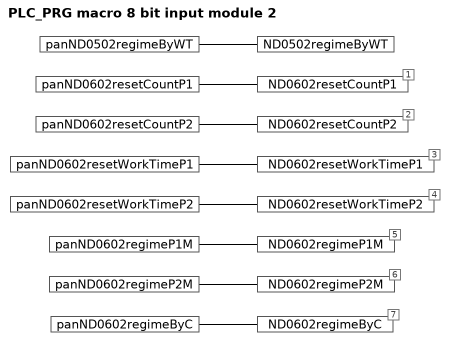
[picture p72: PLC_PRG macro 8 bit input module 2 (CFC)]
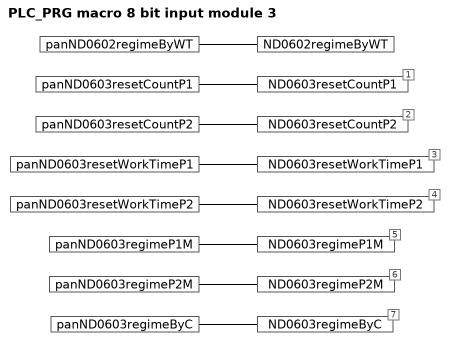
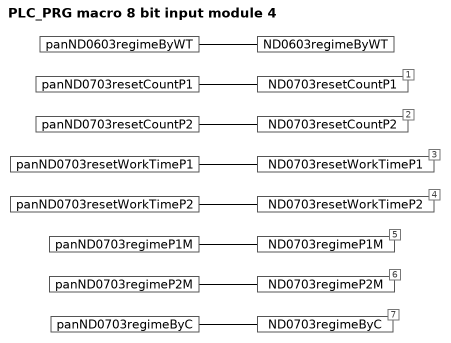
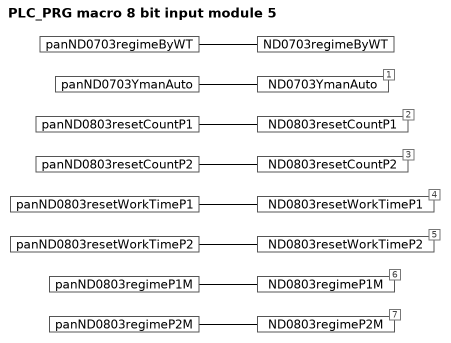
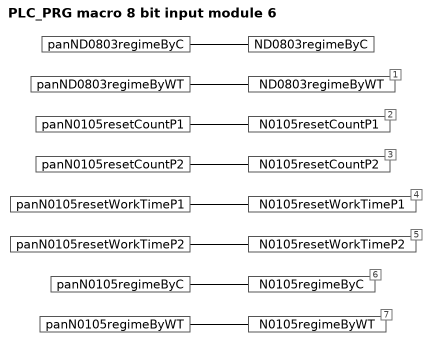
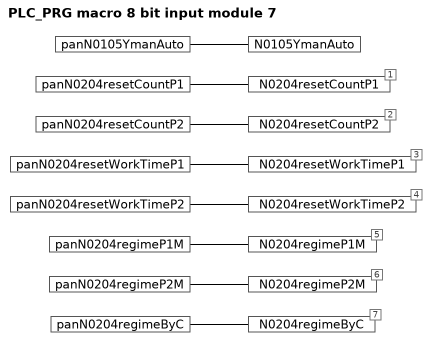
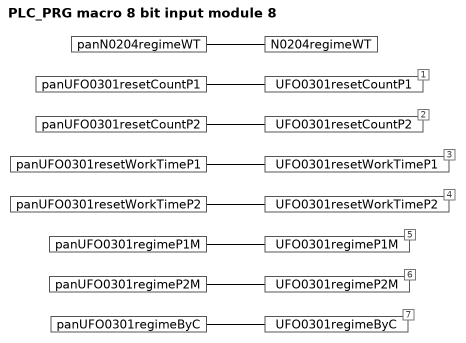
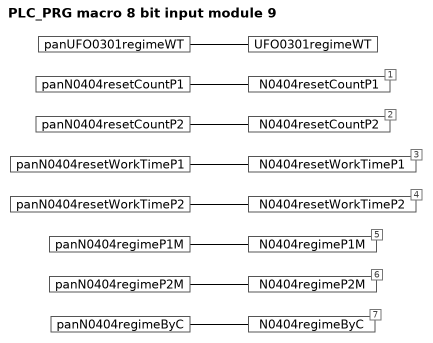
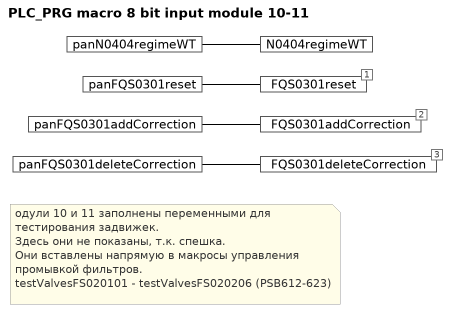
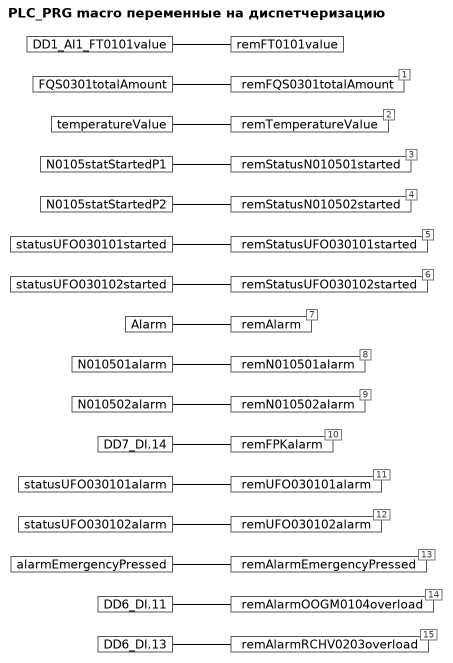
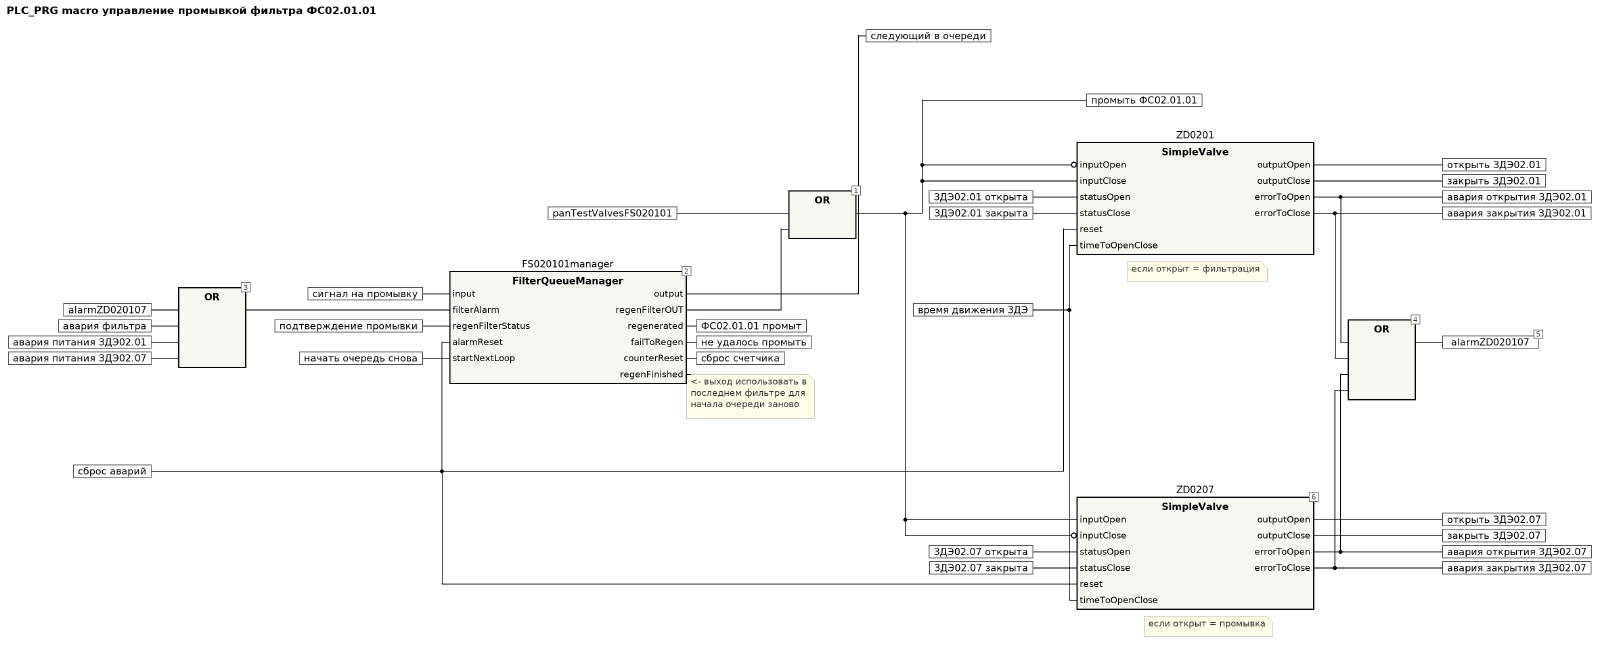
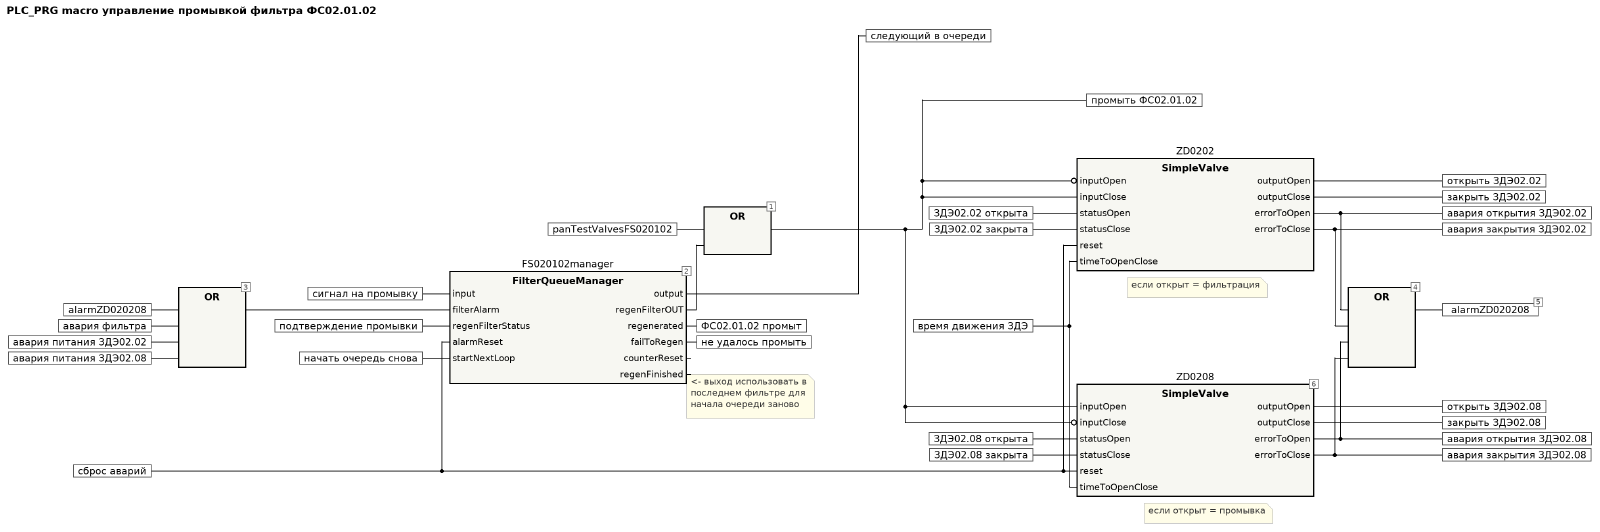
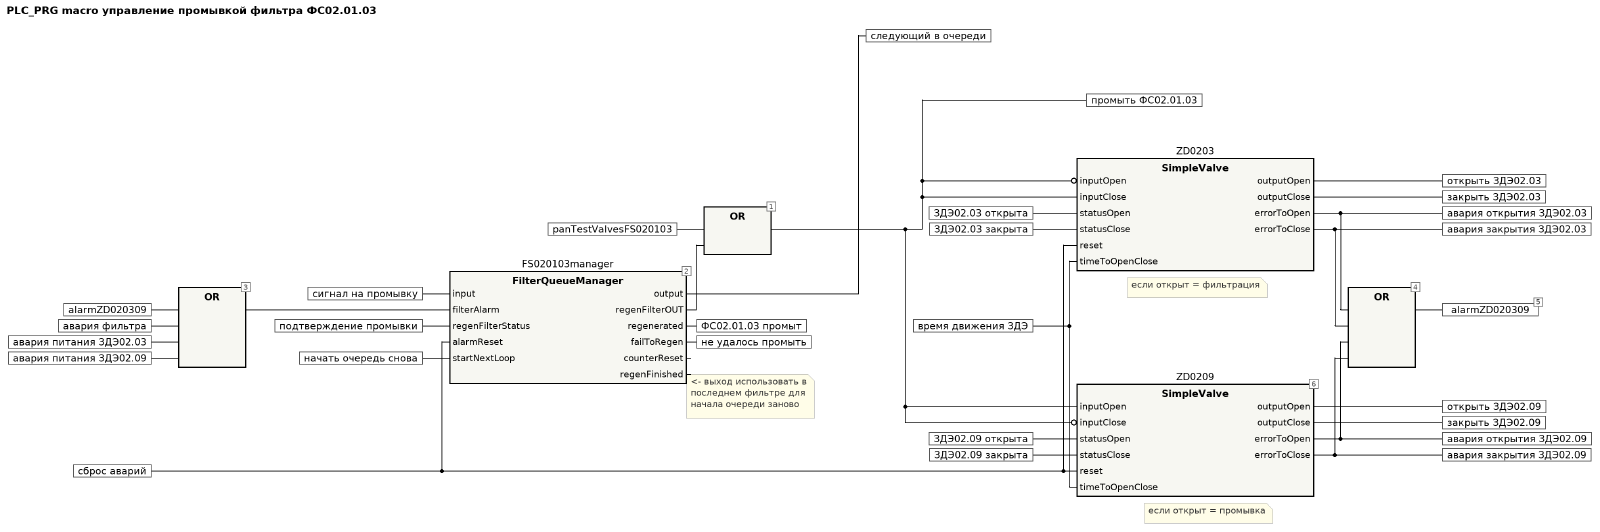
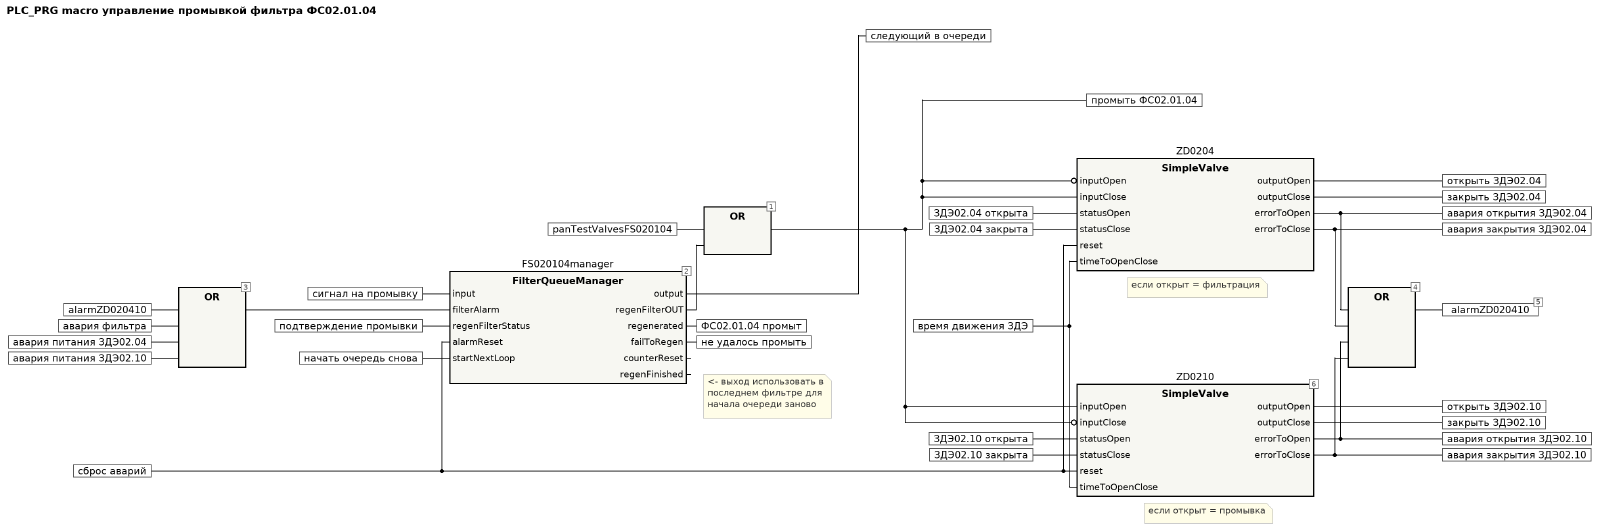
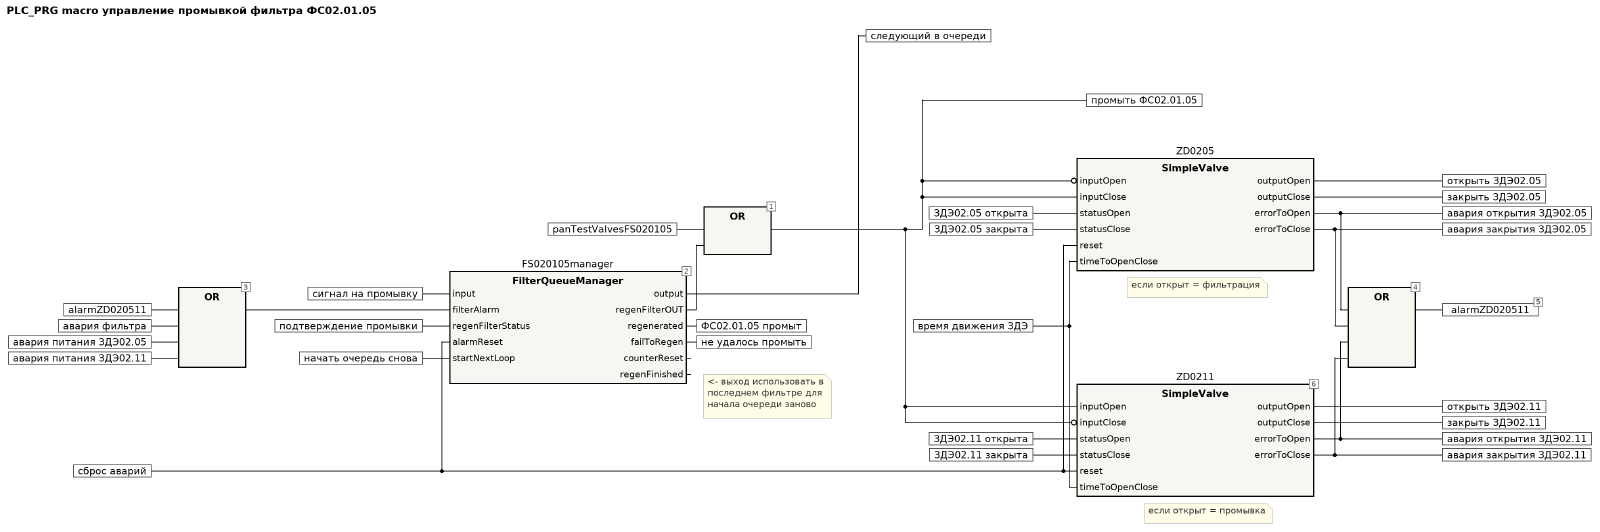
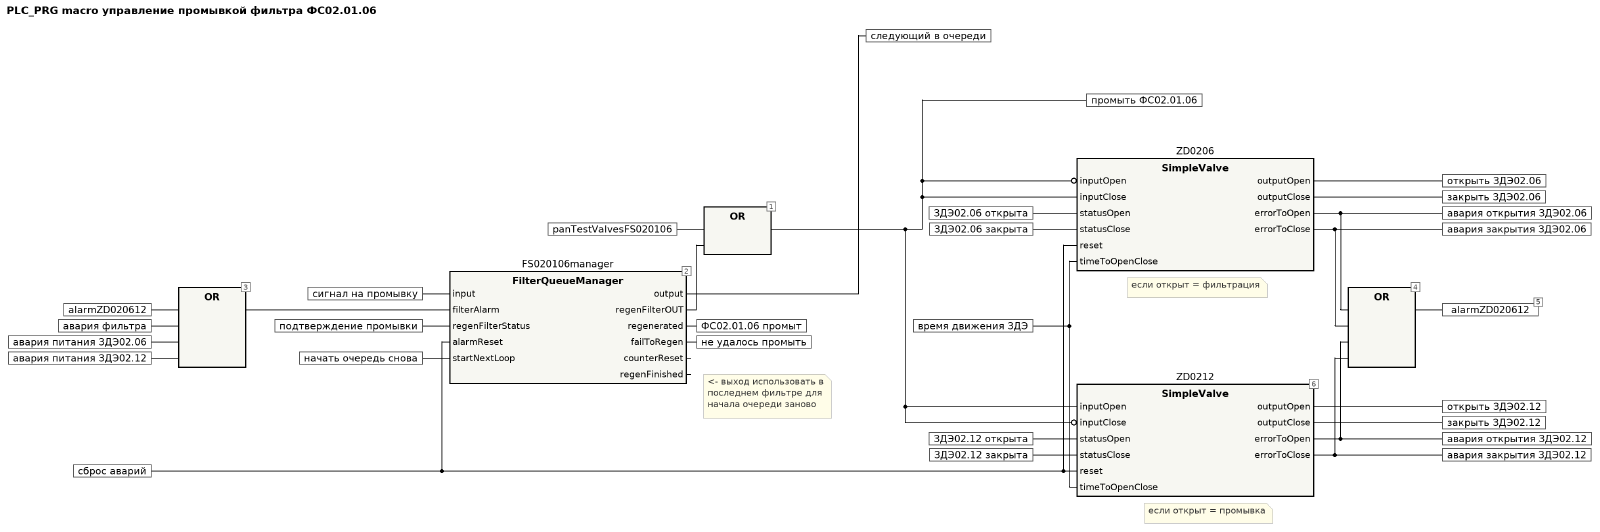
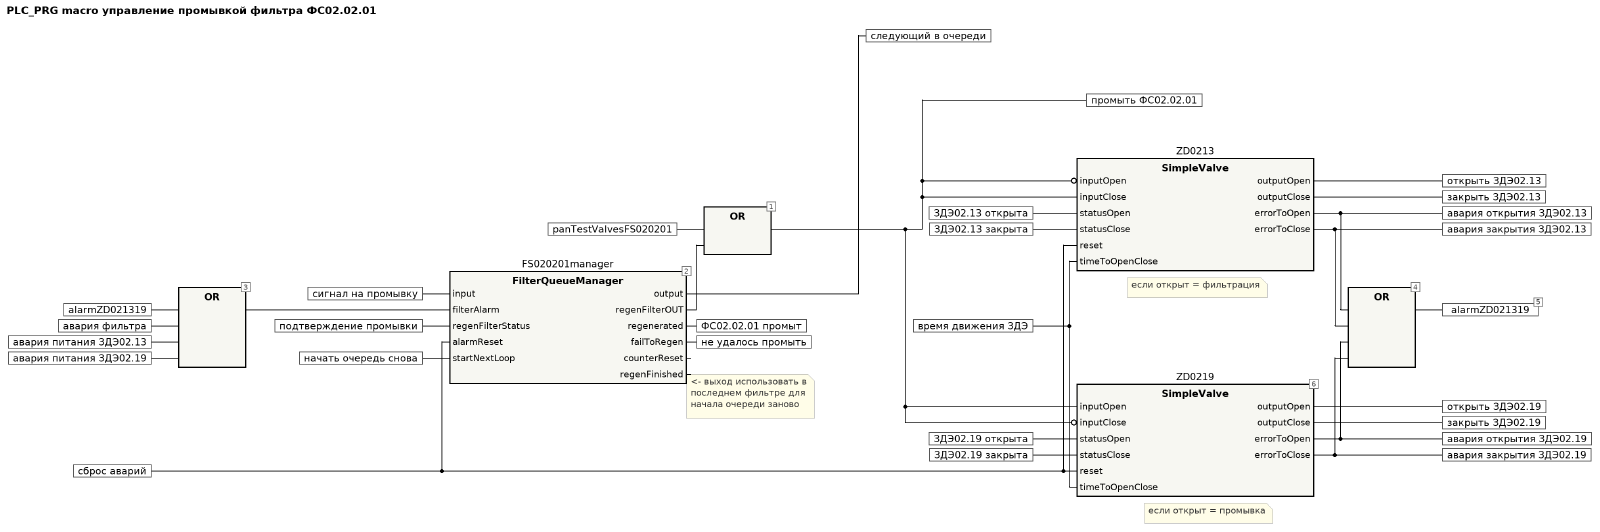
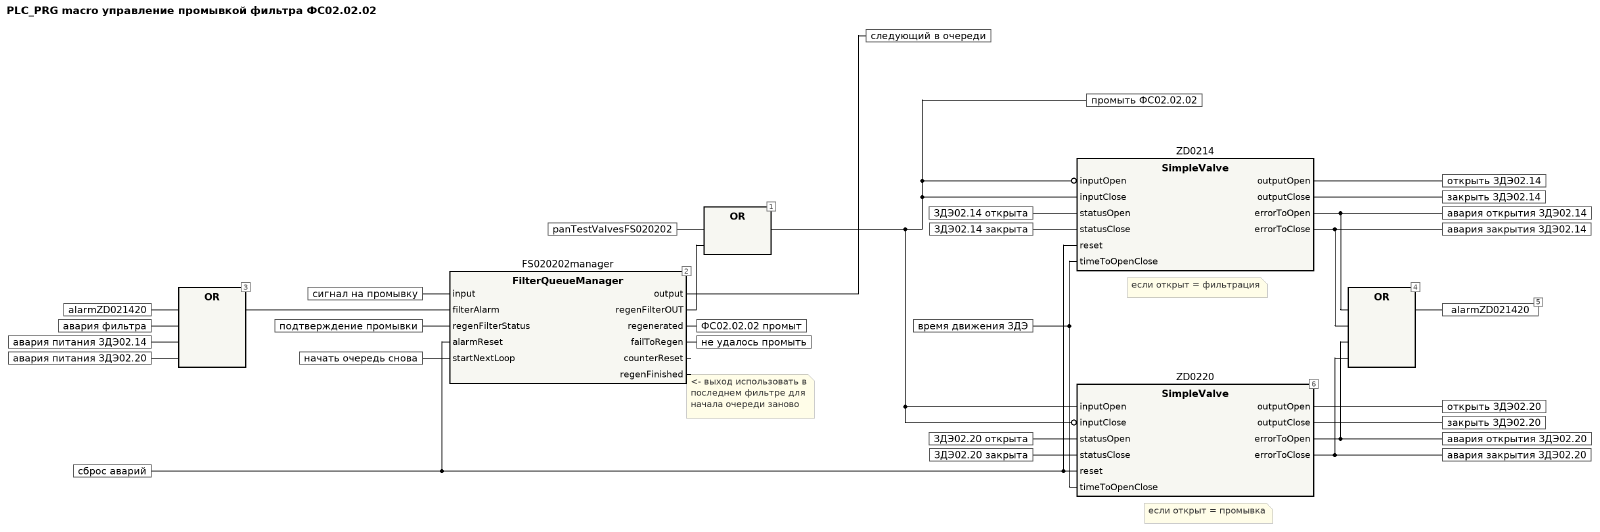
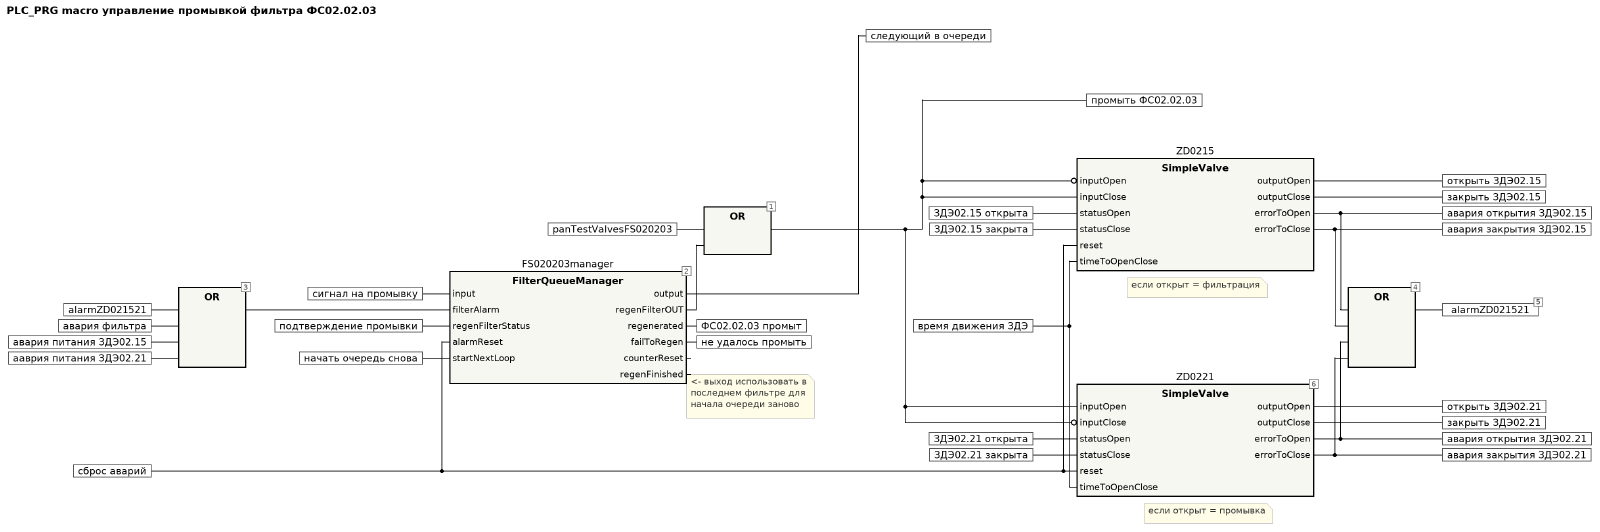
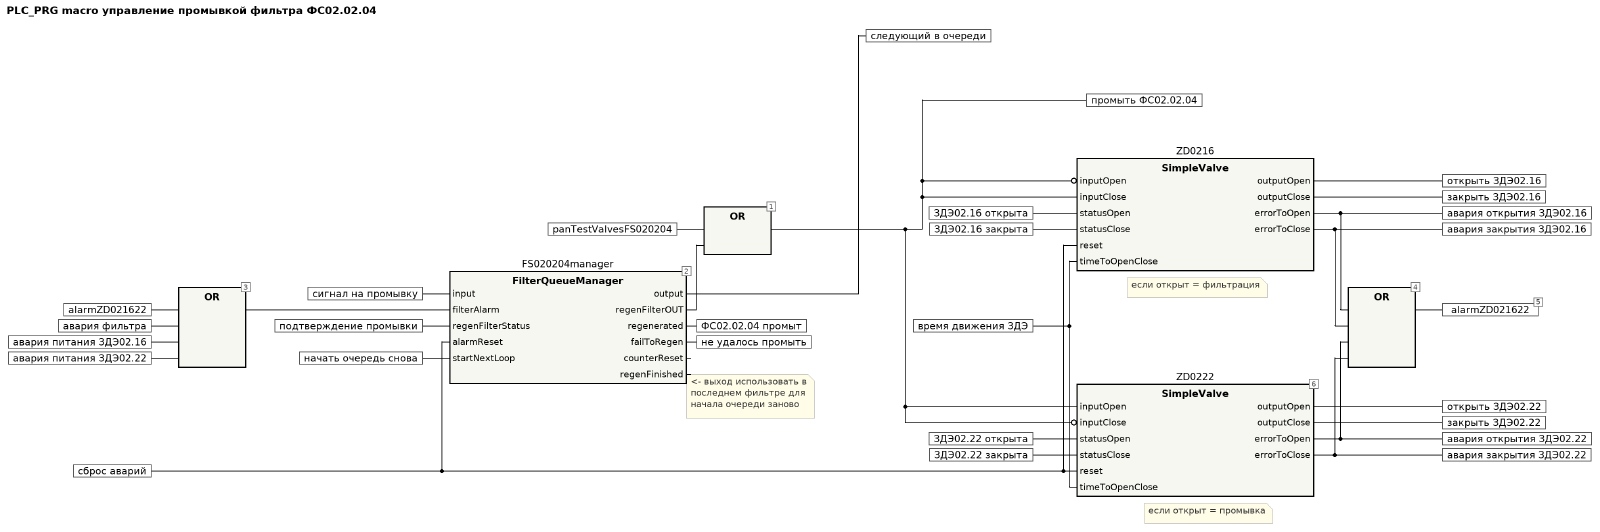
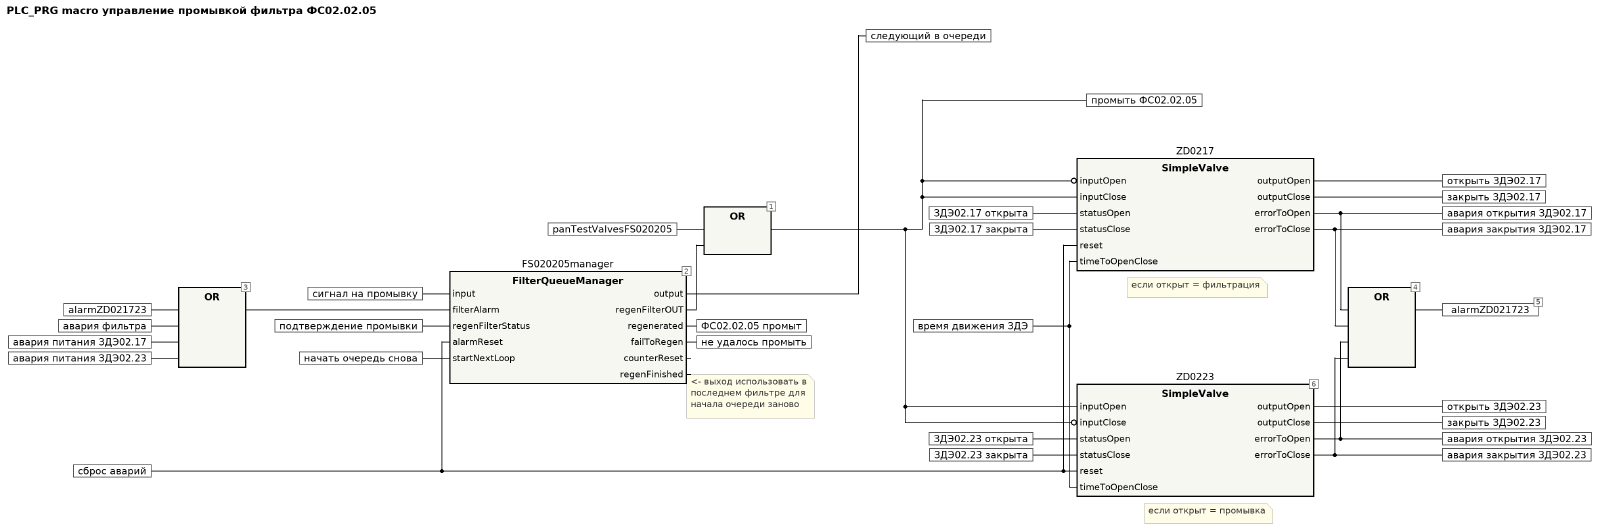
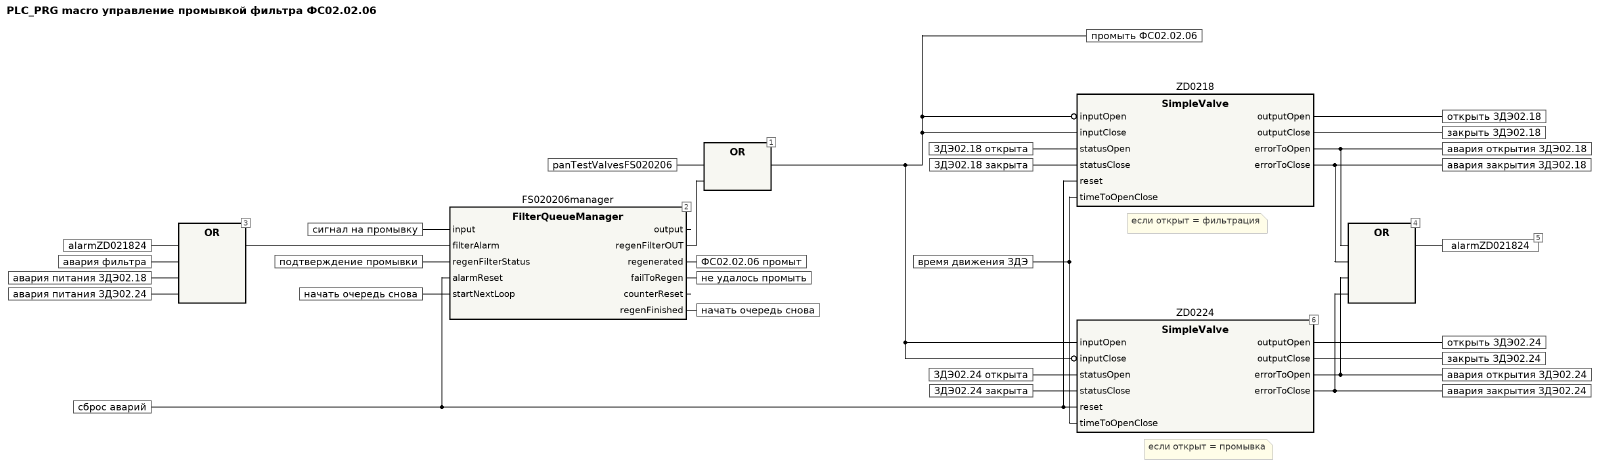
_CFC_ (* Continuous Function Chart, elements in execution order *)
(* в этом макросе лежит управление режимом тестирования задвижек ЗДЭ03 / Тестирование запрещает автоматический запуск УФО от ПЛК *)
(* 1=открыть; 0 = закрыть *)
(* авария питания КШЭ04.01 *)
(* авария НД05.02/02 *)
(* авария НД05.02/01 *)
(* инвертирование сигнала, чтобы все аварии / обозначались как 1 (TRUE) *)
(* авария питания ЗДЭ02.24 *)
(* авария питания ЗДЭ02.23 *)
(* авария питания ЗДЭ02.22 *)
(* авария питания ЗДЭ02.21 *)
(* авария питания ЗДЭ02.20 *)
(* авария питания ЗДЭ02.19 *)
(* авария питания ЗДЭ02.18 *)
(* авария питания ЗДЭ02.17 *)
(* авария питания ЗДЭ02.16 *)
(* авария питания ЗДЭ02.15 *)
(* авария питания ЗДЭ02.14 *)
(* авария питания ЗДЭ02.13 *)
(* авария питания ЗДЭ02.12 *)
(* авария питания ЗДЭ02.11 *)
(* авария питания ЗДЭ02.10 *)
(* авария питания ЗДЭ02.09 *)
(* авария питания ЗДЭ02.08 *)
(* авария питания ЗДЭ02.07 *)
(* авария питания ЗДЭ02.06 *)
(* авария питания ЗДЭ02.05 *)
(* авария питания ЗДЭ02.04 *)
(* авария питания ЗДЭ02.03 *)
(* авария питания ЗДЭ02.02 *)
(* авария питания ЗДЭ02.01 *)
(* очередь передается на 2 ступень *)
(* подсчет общего объема стоков, прошедшего через расходомер FT01.02 *)
(* сброс счетчика стоков до следующей промывки *)
(* авария (при 0) ФС02.02/01 *)
(* авария (при 0) ФС02.02/02 *)
(* авария (при 0) ФС02.02/03 *)
(* авария (при 0) ФС02.02/04 *)
(* авария (при 0) ФС02.02/05 *)
(* авария (при 0) ФС02.02/06 *)
(* авария (при 0) ФС02.01/01 *)
(* авария (при 0) ФС02.01/02 *)
(* авария (при 0) ФС02.01/03 *)
(* авария (при 0) ФС02.01/04 *)
(* авария (при 0) ФС02.01/05 *)
(* авария (при 0) ФС02.01/06 *)
(* 0=авария *)
(* заданный до промывки объем *)
(* текущий объем *)
(* Пуск Н02.04/02 *)
(* Пуск Н02.04/01 *)
(* Стоп Н02.04 *)
(* Сухой ход Н02.04 (LS02.03) 0=сух.ход *)
(* Клапан КЭМ08.01 открыт. *)
(* Клапан КЭМ07.01 открыт. *)
(* Клапан КЭМ06.01 открыт. *)
(* Клапан КЭМ05.01 открыт. *)
(* промывка ФС02.02/01 *)
(* промывка ФС02.02/02 *)
(* промывка ФС02.02/03 *)
(* промывка ФС02.02/04 *)
(* промывка ФС02.02/05 *)
(* промывка ФС02.02/06 *)
(* Авария Н02.04/02 (0=авария) *)
(* Авария Н02.04/01 (0=авария) *)
(* импульсный расходомер *)
(* авария Н04.04/02, 0=авария *)
(* авария Н04.04/01, 0=авария *)
(* сухой ход Н04.04, 0=защита *)
(* авт.пуск Н04.04 *)
(* пуск Н04.04/01 *)
(* пуск Н04.04/02 *)
(* стоп Н04.04 *)
(* подающий насос ФПК работает *)
(* статус КШЭ04.01 закрыт *)
(* Закрыть КШЭ04.01 *)
(* статус КШЭ04.01 открыт *)
(* Открыть КШЭ04.01 *)
(* авария ФПК *)
(* Авария входа AI6 ПЛК, давл.ФПК *)
(* Давление на входе ФПК / 0...16 бар (мах допуст.10) *)
(* LSА02.01 Перелив РЧВ02.03 *)
(* авария питания ЗДЭ02.25 *)
(* термоконтакт Н01.05/02 *)
(* термоконтакт Н01.05/01 *)
(* Авария ЧРП Н01.05 *)
(* КМ3 питание насоса 2 *)
(* КМ2 питание насоса 1 *)
(* КМ1 питание ЧРП *)
(* Пуск  Н01.05 *)
(* время на создание потока *)
(* Стоп  Н01.05 (сброс самоподхвата реле) *)
(* SA1 Ручной выбор Н01.05/02 = главный *)
(* SA1 Ручной выбор Н01.05/01 = главный *)
(* LS01.04 - нижний уровень ОГМ01.04, сухой ход Н01.05 *)
(* LS01.03 - рабочий верхний уровень ОГМ01.04 автоматический пуск 01.05 *)
(* Статус ПУСК ЧРП Н01.05 *)
(* Инициализирует требуемые булевые переменные / в момент старта выполнения программы. *)
(* LSA01.02 перелив ОГМ01.04 *)
(* сухой ход НД08.03/02 *)
(* сухой ход НД08.03/01 *)
(* сухой ход НД08.03/02 *)
(* сухой ход НД08.03/01 *)
(* авария входа рН-метра QE01.02 *)
(* рН-метр QE01.01 на входе, / диапазон 0...14 *)
(* расходомер FT01.02 на входе, / диапазон 0...600куб/час *)
(* авария входа расходомера FT01.01 *)
(* управление 4...20мА НД08.04 *)
(* пуск/стоп НД08.04 *)
(* насос Н04.01 работает *)
(* авария НД08.04 *)
(* авария привода НД08.03/02 *)
(* авария привода НД08.03/01 *)
(* АВАРИИ *)
(* управление 4...20мА НД05.02/02 *)
(* пуск/стоп НД05.02/02 *)
(* авария НД05.02/02 *)
(* авария НД05.02/01 *)
(* пуск/стоп НД05.02/01 *)
(* управление 4...20мА НД05.02/01 *)
(* датчик температуры в помещении / (метран) диапазон: 0...+100С *)
(* лампа АВАРИЯ *)
(* авария входа датчика температуры *)
(* ошибка блока дозирования НД05.02 *)
(* авария НД06.02/02 *)
(* авария НД06.02/01 *)
(* управление 4...20мА НД06.02/02 *)
(* пуск/стоп НД06.02/02 *)
(* пуск/стоп НД06.02/01 *)
(* управление 4...20мА НД06.02/01 *)
(* авария НД06.03/02 *)
(* авария НД06.03/01 *)
(* управление 4...20мА НД06.03/02 *)
(* пуск/стоп НД06.03/02 *)
(* пуск/стоп НД06.03/01 *)
(* управление 4...20мА НД06.03/01 *)
(* авария НД06.02/02 *)
(* авария НД06.02/01 *)
(* авария НД06.03/02 *)
(* авария НД06.03/01 *)
(* авария НД07.03/02 *)
(* авария НД07.03/01 *)
(* пуск/стоп НД07.03/02 *)
(* пуск/стоп НД07.03/01 *)
(* управление 4...20мА НД07.03/02 *)
(* управление 4...20мА НД07.03/01 *)
(* авария НД07.03/02 *)
(* авария НД07.03/01 *)
(* авария привода НД08.03/02 *)
(* авария привода НД08.03/01 *)
(* управление 4...20мА НД08.03/02 *)
(* пуск/стоп НД08.03/02 *)
(* пуск/стоп НД08.03/01 *)
(* управление 4...20мА НД08.03/01 *)
(* авария НД08.04 *)
(* расходомер FT01.01 на входе, / диапазон 0...600куб/час *)
(* авария входа расходомера FT01.02 *)
(* авария входа рН-метра QE01.01 *)
(* рН-метр QE01.02 на входе, / диапазон 0...14 *)
(* ФПК не запустился *)
(* ФПК готов к приему *)
(* подающий насос ФПК работает *)
(* авария ФПК *)
(* Давление на входе ФПК (0...16 бар) *)
(* датчик уровня осадка *)
(* Защита от сухого хода насоса ФПК *)
(* запуск фильтрации *)
(* время работы ФПК после спада сигнала датч.осадка *)
(* время контроля старта ФПК (по умолч.=3мин) *)
(* авария Н04.04/02 *)
(* авария Н04.04/01 *)
(* авария УФО03.01/01 *)
(* авария УФО03.01/02 *)
(* работа УФО03.01/01 *)
(* Для подачи предостережения на пульте / оператора (при необходимости), а также / сигнализации лампой АВАРИЯ. *)
(* авария УФО03.01/01 *)
(* работа УФО03.01/02 *)
(* авария УФО03.01/02 *)
(* Контроль, если УФО включили вручную, / а потока при этом нет. *)
(* работа М06.04 (УПК) *)
(* работа М07.02 (УПЩ) *)
(* работа М08.02 (УПФ) *)
(* авария М06.04 (УПК) *)
(* авария М07.02 (УПЩ) *)
(* авария М08.02 (УПФ) *)
(* пуск/стоп НД07.03/02 *)
(* пуск/стоп НД07.03/01 *)
(* пуск/стоп НД08.04 *)
(* пуск/стоп НД06.02/02 *)
(* пуск/стоп НД06.02/01 *)
(* пуск/стоп НД06.03/02 *)
(* пуск/стоп НД06.03/01 *)
(* пуск/стоп НД08.03/02 *)
(* пуск/стоп НД08.03/01 *)
(* промывка ФС02.01/01 *)
(* промывка ФС02.01/02 *)
(* промывка ФС02.01/03 *)
(* промывка ФС02.01/04 *)
(* промывка ФС02.01/05 *)
(* промывка ФС02.01/06 *)
(* Авария Н02.04/02 (0=авария) *)
(* Авария Н02.04/01 (0=авария) *)
(* здесь мгновенный расход / в кубометрах в час (FT01.02) *)
(* выдает импульс / каждую секунду *)
(* если есть расход / (больше нуля) *)
(* преобразуем расход из / кубометров в час в / кубометры в секунду *)
(* суммируем каждую секунду значение / мгновенного расхода в кубометрах в секунду *)
(* блок подачи сигнала на промывку *)
(* авария КНС *)
(* Авария питания розеток / управл.клапанов фильтров. *)
(* Авария питания клапанов КЭМ. *)
(* авария сети (РКФ) *)
(* Блок управления разрешением работы КНС *)
(* Нажат аварийный стоп. *)
(* разрешение работы КНС / 1 = разрешено *)
(* авария сети (РКФ) *)
(* Нажат аварийный стоп. *)
(* LSA01.02 перелив ОГМ01.04 *)
(* контроль обрыва или ошибок модулей в сети ПЛК *)
(* вкл КМ2 *)
(* статус-пуск Н01.05/01 *)
(* Статус ПУСК / ЧРП Н01.05 *)
(* вкл КМ3 *)
(* статус-пуск Н01.05/02 *)
(* авария питания ЗДЭ03.01 *)
(* авария питания ЗДЭ03.02 *)
(* авария обоих УФО, если проблемы / открытия/закрытия на одной из задвижек *)
(* 0 = перелив *)
#0 rTrigStartInitializer:R_TRIG(CLK: TRUE)
#1 startInitializer <= #0.Q
#2 MACRO контроль температуры в помещении(pin 1 "вход датчика температуры": DD1_AI0, pin 2 "минимально допустимая температура в помещении": maxTemperature, pin 3 "максимально допустимая температура в помещении": minTemperature)
	(* не смотрим конкретный тип ошибки / (работает не точно, обрыв определяет как слишком маленькое значение) / если не равно 0 - значит на входе ошибка *)
	(* задаем границы допустимой температуры в помещении / проверяем что измеренное значение в заданном диапазоне *)
	#3 DD1_AI0_temperature:DECODE_FLOAT(VALUE: pin 1, DEF_VALUE: -)
	#4 NE(#3._ERR, 0)
	out 2 "авария датчика температуры" <= #4
	out 1 "температура в помещении" <= #3.OUT_VALUE
	#5 REAL_TO_INT(#3.OUT_VALUE)
	#6 temperatureLimits:LIMITALARM(IN: #5, HIGH: pin 3, LOW: pin 2)
	out 3 "температура выше заданного диапазона" <= #6.O
	out 4 "температура ниже заданного диапазона" <= #6.U
	#7 temperatureLimits:LIMITALARM(IN: -, HIGH: -, LOW: -)
END_MACRO
#8 temperatureValue <= #2.out 1
#9 DD1_AI0_error <= #2.out 2
#10 alarmHighTemperature <= #2.out 3
#11 alarmLowTemperature <= #2.out 4
#12 OR(testKSHE0401, DD7_DI.13)
#13 MACRO клапан шаровый перед ФПК (КШЭ04.01)(pin 1 "сигнал "подающий насос ФПК" работает": #12, pin 2 "статус КШЭ04.01 открыт": DD9_DI.2, pin 3 "статус КШЭ04.01 закрыт": DD9_DI.3, pin 4 "сброс аварий": alarmReset, pin 5 "время на открытие/закрытие": timeToOpenCloseValve)
	#14 FPKkshe0401DelayToOpen:TON(IN: #16.outputOpen, PT: T#1s)
	out 1 "выход на открытие КШЭ04.01" <= #14.Q
	#15 FPKkshe0401DelayToClose:TON(IN: #16.outputClose, PT: T#1s)
	out 2 "выход на закрытие КШЭ04.01" <= #15.Q
	#16 FPKkshe0401:SimpleValve(inputOpen: pin 1, inputClose: #17, statusOpen: pin 2, statusClose: pin 3, reset: pin 4, timeToOpenClose: pin 5)
	#17 NOT(pin 1)
	out 3 "авария на открытие КШЭ04.01" <= #16.errorToOpen
	out 4 "авария на закрытие КШЭ04.01" <= #16.errorToClose
END_MACRO
#18 DD4_DO.2 <= #13.out 1
#19 DD4_DO.3 <= #13.out 2
#20 FPKkshe0401errorToOpen <= #13.out 3
#21 FPKkshe0401errorToClose <= #13.out 4
#22 OR(DD1_AI0_error, DD1_AI1_error, DD1_AI2_error, DD1_AI3_error, DD1_AI4_error, alarmHighTemperature, alarmLowTemperature, ND0502dosingError, ND0602dosingError, ND0603dosingError, ND0803dosingError, ND0804dosingError, DD1_DI6, DD1_DI7, N010501alarm, N010502alarm, ZDE0225errorToOpen, ZDE0225errorToClose, DD7_DI.14, FPKnotStarted, DD1_AI5_error, FPKkshe0401errorToOpen, FPKkshe0401errorToClose, DD5_DI.27, DD5_DI.29, filterFailToRegen020101, errorToOpenZD0201, errorToCloseZD0201, errorToOpenZD0207, errorToCloseZD0207, filterFailToRegen020102, errorToOpenZD0202, errorToCloseZD0202, errorToOpenZD0208, errorToCloseZD0208, filterFailToRegen020103, errorToOpenZD0203, errorToCloseZD0203, errorToOpenZD0209, errorToCloseZD0209, filterFailToRegen020104, errorToOpenZD0204, errorToCloseZD0204, errorToOpenZD0210, errorToCloseZD0210, filterFailToRegen020105, errorToOpenZD0205, errorToCloseZD0205, errorToOpenZD0211, errorToCloseZD0211, filterFailToRegen020106, errorToOpenZD0206, errorToCloseZD0206, errorToOpenZD0212, errorToCloseZD0212, filterFailToRegen020201, errorToOpenZD0213, errorToCloseZD0213, errorToOpenZD0219, errorToCloseZD0219, filterFailToRegen020202, errorToOpenZD0214, errorToCloseZD0214, errorToOpenZD0220, errorToCloseZD0220, filterFailToRegen020203, errorToOpenZD0215, errorToCloseZD0215, errorToOpenZD0221, errorToCloseZD0221, filterFailToRegen020204, errorToOpenZD0216, errorToCloseZD0216, errorToOpenZD0222, errorToCloseZD0222, filterFailToRegen020205, errorToOpenZD0217, errorToCloseZD0217, errorToOpenZD0223, errorToCloseZD0223, filterFailToRegen020206, errorToOpenZD0218, errorToCloseZD0218, errorToOpenZD0224, errorToCloseZD0224, alarmPLKnetwork, alarmND050201, alarmND050202, alarmND060201, alarmND060202, alarmND060301, alarmND060302, alarmND070301, alarmND070302, alarmND080301, alarmND080302, alarmND0804, alarmOGM0104overload, alarmRCHV0203overload, alarmN040402, alarmN040401, alarmM0604, alarmM0702, alarmM0802, alarmN020401, alarmN020402, alarmFS020101, alarmFS020102, alarmFS020103, alarmFS020104, alarmFS020105, alarmFS020106, alarmFS020201, alarmFS020202, alarmFS020203, alarmFS020204, alarmFS020205, alarmFS020206, alarmZDE0201power, alarmZDE0202power, alarmZDE0203power, alarmZDE0204power, alarmZDE0205power, alarmZDE0206power, alarmZDE0207power, alarmZDE0208power, alarmZDE0209power, alarmZDE0210power, alarmZDE0211power, alarmZDE0212power, alarmZDE0213power, alarmZDE0214power, alarmZDE0215power, alarmZDE0216power, alarmZDE0217power, alarmZDE0218power, alarmZDE0219power, alarmZDE0220power, alarmZDE0221power, alarmZDE0222power, alarmZDE0223power, alarmZDE0224power, alarmZDE0225power, alarmKSHE0401power, alarmKNS, alarmPowerSocketFS, alarmKEMvalvesPower, alarmEmergencyPressed, alarmRKF, errorToOpenZDE0301, errorToCloseZDE0301, errorToOpenZDE0302, errorToCloseZDE0302, alarmZDE0301power, alarmZDE0302power)
#23 DD1_DO11 <= #22
#24 alarm <= #22
#25 MACRO контроль аналогового входа DD1_AI1(pin 1 "вход": DD1_AI1)
	(* Не смотрим конкретную ошибку, / определяем,что вход неисправен без расшифровки. *)
	#26 DD1_AI1_FT0101:DECODE_FLOAT(VALUE: pin 1, DEF_VALUE: -)
	#27 NE(#26._ERR, 0)
	out 2 "авария" <= #27
	out 1 "выход" <= #26.OUT_VALUE
END_MACRO
#28 DD1_AI1_FT0101value <= #25.out 1
#29 DD1_AI1_error <= #25.out 2
#30 MACRO контроль аналогового входа DD1_AI2(pin 1 "вход": DD1_AI2)
	(* Не смотрим конкретную ошибку, / определяем,что вход неисправен без расшифровки. *)
	#31 DD1_AI2_FT0102:DECODE_FLOAT(VALUE: pin 1, DEF_VALUE: -)
	#32 NE(#31._ERR, 0)
	out 2 "авария" <= #32
	out 1 "выход" <= #31.OUT_VALUE
END_MACRO
#33 DD1_AI2_FT0102value <= #30.out 1
#34 DD1_AI2_error <= #30.out 2
#35 MACRO управление Н01.05 (поддержание заданного расхода по FT01.02)(pin 1 "статус ПУСК ЧРП (реле)": DD5_DI.4, pin 2 "LS01.03 раб.уров.": DD6_DI.12, pin 3 "LS01.04 ниж.уров.(сух.ход)": DD5_DI.0, pin 4 "SA1ручной выб.Н01.05/01-главный": DD5_DI.5, pin 5 "SA1ручной выб.Н01.05/02-главный": DD5_DI.6, pin 6 "включить режим "по кол.вкл."": N0105regimeByC, pin 7 "включить режим "по наработке"": N0105regimeByWT, pin 8 "значение расхода от FT01.02": DD1_AI2_FT0102value, pin 9 "уставка расхода": N0105flowSetValue, pin 10 "время на создание потока": N0105minFlowTime, pin 11 "Р-коэфф.": N0105koeffP, pin 12 "I-коэфф": N0105koeffI, pin 13 "Д-коэфф": N0105koeffD, pin 14 "управление ЧРП в ручн.реж.(4...20мА)": N0105YoutManual, pin 15 "переключатель управление ЧРП РУЧН/АВТ": N0105YmanAuto, pin 16 "мин.допустимый расход": N0105minFlow, pin 17 "термоконтакт Н01.05/01": DD5_DI.2, pin 18 "термоконтакт Н01.05/02": DD5_DI.3, pin 19 "авария ЧРП Н01.05": DD5_DI.1, pin 20 "сброс аварии": alarmReset, pin 21 "сброс кол-ва вкл.Н01.05/01": N0105resetCountP1, pin 22 "сброс кол-ва вкл.Н01.05/02": N0105resetCountP2, pin 23 "сброс наработки Н01.05/01": N0105resetWorkTimeP1, pin 24 "сброс наработки Н01.05/02": N0105resetWorkTimeP2)
	(* Если насос создает давление меньше / указанного, то авария. *)
	(* если на входе true / то нижнее значение, / иначе то, что посередине *)
	(* по умолчанию при старте программы *)
	(* управление Н01.05 - поддержание / заданного расхода по FT01.02 *)
	(* режимы по количеству включений,  или по наработке / активны если оба входа SA1 не активны *)
	(* Пуск  Н01.05 *)
	(* время на создание потока *)
	#36 OR(pin 2, #37.Q)
	#37 N0105startTrig:R_TRIG(CLK: pin 1)
	#38 N0105stopTrig:F_TRIG(CLK: pin 1)
	#39 N0105startTrigg:RS(SET: #36, RESET1: #42)
	#40 N0105regime:choosePumpRegime(start: #39.Q1, pump1Main: pin 4, pump2Main: pin 5, byCounter: #49, byWorkTime: #54)
	out 2 "статус режим "Н01.05/01 - главный"" <= #40.pump1MainActive
	out 3 "статус режим "Н01.05/02 - главный"" <= #40.pump2MainActive
	#41 AND(#53.pump1active, #63)
	out 4 "статус режим "по кол-ву вкл."" <= #40.byCounterActive
	out 15 "авария Н01.05/01" <= #45.Q1
	#42 OR(#38.Q, #43)
	out 5 "статус режим "по наработке"." <= #40.byWorkTimeActive
	#43 NOT(pin 3)
	#44 OR(#41, #48, NOT pin 17)
	#45 N010501alarmTrig:RS(SET: #44, RESET1: pin 20)
	#46 N010501alarm <= #45.Q1
	#47 NOT(#39.Q1)
	out 1 "СТОП (сброс самоподхвата реле пуска ЧРП)." <= #47
	#48 AND(#53.pump1active, NOT pin 19)
	#49 AND(NOT pin 4, NOT pin 5, #52.Q1)
	#50 OR(pin 6, startInitializer)
	#51 N0105regByCinit:R_TRIG(CLK: #50)
	#52 N0105regByCtrig:RS(SET: #51.Q, RESET1: #55.Q)
	#53 N0105twoPumpOneDriveManager:TwoPumpOneDriveManager(startStopPump1: #40.startPump1, startStopPump2: #40.startPump2, alarmPump1: N010501alarm, alarmPump2: N010502alarm, alarmReset: alarmReset, counterStart: #40.startByCounter, Pump1ResetCounter: pin 21, Pump2ResetCounter: pin 22, ValueToResetCounter: -, workTimeStart: #40.startByWorkTime, workTimePump1Reset: pin 23, workTimePump2Reset: pin 24, timeKM1off: -, timeKM23DelayON: -, timeKM23offDelay: -, timeReadyToStartDelay: -)
	out 6 "кол-во включений Н01.05/01" <= #53.counterPump1
	out 7 "кол-во включений Н01.05/02" <= #53.counterPump2
	out 8 "наработка Н01.05/01" <= #53.currentWorkTimePump1
	#54 AND(NOT pin 4, NOT pin 5, #56.Q1)
	out 9 "наработка Н01.05/02" <= #53.currentWorkTimePump2
	out 10 "КМ1-питание ЧРП" <= #53.DriveKM
	#55 N0105regWTinit:R_TRIG(CLK: pin 7)
	#56 N0105regWTtrig:RS(SET: #55.Q, RESET1: #51.Q)
	out 11 "КМ2-питание Н01.05/01" <= #53.pump1KM
	out 12 "КМ3-питание Н01.05/02" <= #53.pump2KM
	out 13 "пуск ЧРП (Н01.05)" <= #53.driveStart
	out 16 "авария Н01.05/02" <= #59.Q1
	#57 AND(NOT pin 19, #53.pump2active)
	#58 OR(#57, #61, NOT pin 18)
	#59 N010502alarmTrig:RS(SET: #58, RESET1: pin 20)
	#60 N010502alarm <= #59.Q1
	#61 AND(#53.pump2active, #63)
	#62 N0105timerminFlow:TON(IN: #53.driveStart, PT: pin 10)
	#63 AND(#62.Q, #64)
	#64 LE(pin 8, pin 16)
	#65 SEL(#53.driveStart, 0, #66.Y)
	out 14 "управление ЧРП (4...20мА)" <= #65
	#66 N0105pidReg:PID(ACTUAL: pin 8, SET_POINT: pin 9, KP: pin 11, TN: pin 12, TV: pin 13, Y_MANUAL: pin 14, Y_OFFSET: -, Y_MIN: 4, Y_MAX: 20, MANUAL: pin 15, RESET: #66.OVERFLOW)
END_MACRO
#67 DD4_DO.13 <= #35.out 1
#68 N0105statRegimeP1M <= #35.out 2
#69 N0105statRegimeP2M <= #35.out 3
#70 N0105statRegimeByC <= #35.out 4
#71 N0105statRegimeByWT <= #35.out 5
#72 N0105counterP1 <= #35.out 6
#73 N0105counterP2 <= #35.out 7
#74 N0105workTimeP1 <= #35.out 8
#75 N0105workTimeP2 <= #35.out 9
#76 DD2_DO.0 <= #35.out 10
#77 DD2_DO.1 <= #35.out 11
#78 DD2_DO.2 <= #35.out 12
#79 DD1_DO0 <= #35.out 13
#80 DD1_AO0 <= #35.out 14
#81 N010501alarm <= #35.out 15
#82 N010502alarm <= #35.out 16
#83 MACRO Сигналы работы с ФП04.02 (фильтр-пресс)(pin 1 "датчик уровня осадка": DD7_DI.15, pin 2 "время работы ФПК (после выкл.датч.осадка)": FPKtimeToWork, pin 3 "защита от сухого хода": DD6_DI.10, pin 4 "ошибка входа AI (обрыв)": DD1_AI5_error, pin 5 "авария ФПК": DD7_DI.14, pin 6 "фильтр-пресс готов к приему": DD7_DI.12, pin 7 "давление на входе в ФПК": DD1_AI5_FPKpressureValue, pin 8 "мах допустимое давление": FPKmaxPressureValue, pin 9 "подающий насос ФПК работает": DD7_DI.13, pin 10 "время контроля старта ФПК": FPKnotStartedTime, pin 11 "сброс аварий": alarmReset)
	(* Условие сброса сигнала о грязном фильтр-прессе: / 1. Пропал сигнал о готовности ФПК; / 2. Появился сигнал о готовности ФПК. / Это значит, что оператор раздвигал плиты, / чистил и снова сдвигал их. *)
	(* максимально допустимое давление / на входе ФПК *)
	(* Давление на входе ФПК / 0...16 бар (мах допуст.10) *)
	(* Время работы ФПК после / спада сигнала уровня осадка / по умолч.15мин. *)
	(* LES01.01-сигнал датчика уровня осадка ОГМ01.04 / запуск процесса фильтрации *)
	(* LS01.01-нижн.уровень на входе ОГМ01.04 / защита от сух. хода насоса ФПК *)
	(* ФПК готов к приему осадка *)
	#84 FPKneedToCleanResetFtrig:F_TRIG(CLK: FPKneedToCleanReset)
	#85 FPKstartTrig:RS(SET: pin 1, RESET1: #91)
	out 1 "запуск/старт ФПК" <= #85.Q1
	#86 FPKstopTimer:TOF(IN: pin 1, PT: pin 2)
	#87 FPKstopFtrig:F_TRIG(CLK: #86.Q)
	#88 AND(#85.Q1, #89)
	#89 NOT(pin 11)
	#90 AND(#85.Q1, #92.Q, #94)
	out 2 "ФПК не стартовал" <= #90
	#91 OR(#87.Q, pin 4, pin 5, #93, #95, #98.Q1)
	#92 FPKnotStartedTimer:TON(IN: #88, PT: pin 10)
	#93 NOT(pin 3)
	#94 NOT(pin 9)
	#95 NOT(pin 6)
	#96 AND(#85.Q1, #97)
	#97 GE(pin 7, pin 8)
	#98 FPKneedToCleanTrig:RS(SET: #96, RESET1: #84.Q)
	out 3 "ФПК нужно почистить!" <= #98.Q1
	#99 S FPKneedToCleanReset <= #98.Q1
	#100 FPKneedToCleanResetRtrig:R_TRIG(CLK: pin 6)
	#101 R FPKneedToCleanReset <= #100.Q
END_MACRO
#102 DD1_DO10 <= #83.out 1
#103 FPKnotStarted <= #83.out 2
#104 FPKneedToClean <= #83.out 3
#105 MACRO контроль аналогового входа DD1_AI3(pin 1 "вход": DD1_AI3)
	(* Не смотрим конкретную ошибку, / определяем,что вход неисправен без расшифровки. *)
	#106 DD1_AI3_QE0101:DECODE_FLOAT(VALUE: pin 1, DEF_VALUE: -)
	#107 NE(#106._ERR, 0)
	out 2 "авария" <= #107
	out 1 "выход" <= #106.OUT_VALUE
END_MACRO
#108 DD1_AI3_QE0101value <= #105.out 1
#109 DD1_AI3_error <= #105.out 2
#110 MACRO контроль аналогового входа DD1_AI4(pin 1 "вход": DD1_AI4)
	(* Не смотрим конкретную ошибку, / определяем,что вход неисправен без расшифровки. *)
	#111 DD1_AI4_QE0102:DECODE_FLOAT(VALUE: pin 1, DEF_VALUE: -)
	#112 NE(#111._ERR, 0)
	out 2 "авария" <= #112
	out 1 "выход" <= #111.OUT_VALUE
END_MACRO
#113 DD1_AI4_QE0102value <= #110.out 1
#114 DD1_AI4_error <= #110.out 2
#115 MACRO контроль аналогового входа DD1_AI5(pin 1 "вход": DD1_AI5)
	(* Не смотрим конкретную ошибку, / определяем,что вход неисправен без расшифровки. *)
	#116 DD1_AI5_FPK:DECODE_FLOAT(VALUE: pin 1, DEF_VALUE: -)
	#117 NE(#116._ERR, 0)
	out 2 "авария" <= #117
	out 1 "выход" <= #116.OUT_VALUE
END_MACRO
#118 DD1_AI5_FPKpressureValue <= #115.out 1
#119 DD1_AI5_error <= #115.out 2
#120 MACRO управление НД05.02 УПГ(pin 1 "вход расходомера в куб/час": DD1_AI1_FT0101value, pin 2 "max производительность НД в мл/мин": ND0502setMaxDosVal, pin 3 "задание дозирования в мл/куб": ND0502setKoefProp, pin 4 "режим:1 насос главный": ND0502regimeP1M, pin 5 "режим: 2 насос главный": ND0502regimeP2M, pin 6 "режим: по наработке": ND0502regimeByWT, pin 7 "режим: по кол-ву включений": ND0502regimeByC, pin 8 "авария 1 насоса": DD6_DI.0, pin 9 "авария 2 насоса": DD6_DI.1, pin 10 "сброс аварий": alarmReset, pin 11 "сброс счетчика включений 1 насоса": ND0502resetCountP1, pin 12 "сброс ссчетчика включений 2 насоса": ND0502resetCountP2, pin 13 "сброс наработки 1 насоса": ND0502resetWorkTimeP1, pin 14 "сброс наработки 2 насоса": ND0502resetWorkTimeP2)
	(* Если на входе SEL = TRUE, / то нижнее значение, / иначе - то,что посередине. *)
	(* сигнал 4...20мА на НД05.02/01 *)
	(* сигнал 4...20мА на НД05.02/02 *)
	#121 SEL(#128.pump1ON, 4, #122.outputValue)
	out 6 "выход 4...20мА насоса 1" <= #121
	#122 ND0502dosing:DosingPumpProportional(flowValue: pin 1, setMinPumpDosingValue: -, setMaxPumpDosingValue: pin 2, minOutputValue: -, maxOutputValue: -, setKoeffProportionality: pin 3, minFlowToStart: -)
	out 1 "ошибка блока дозирования" <= #122.dosingError
	#123 SEL(#128.pump2ON, 4, #122.outputValue)
	#124 linTrafND050201:LIN_TRAFO(IN: #123, IN_MIN: 4, IN_MAX: 20, OUT_MIN: 0, OUT_MAX: 1000)
	#125 REAL_TO_WORD(#124.OUT)
	out 7 "выход 4...20мА насоса 2" <= #125
	#126 ND0502regime:choosePumpRegime(start: #122.startDosingPump, pump1Main: pin 4, pump2Main: pin 5, byCounter: #127, byWorkTime: pin 6)
	out 2 "статус: 1 насос главный" <= #126.pump1MainActive
	out 3 "статус: 2 насос главный" <= #126.pump2MainActive
	out 4 "статус: по кол-ву включений" <= #126.byCounterActive
	#127 OR(pin 7, startInitializer)
	out 5 "статус: по наработке" <= #126.byWorkTimeActive
	#128 ND0502manager:TwoPumpManager(startStopPump1: #126.startPump1, startStopPump2: #126.startPump2, alarmPump1: #129, alarmPump2: #130, alarmReset: pin 10, counterStart: #126.startByCounter, Pump1ResetCounter: pin 11, Pump2ResetCounter: pin 12, ValueToResetCounter: -, workTimeStart: #126.startByWorkTime, workTimePump1Reset: pin 13, workTimePump2Reset: pin 14)
	out 12 "сигнал на включение насоса 1" <= #128.pump1ON
	#129 NOT(pin 8)
	out 13 "сигнал на включение насоса 2" <= #128.pump2ON
	out 8 "счетчик включений насоса 1" <= #128.counterPump1
	#130 NOT(pin 9)
	out 9 "счетчик включений насоса 2" <= #128.counterPump2
	out 10 "счетчик наработки насоса 1" <= #128.currentWorkTimePump1
	out 11 "счетчик наработки насоса 2" <= #128.currentWorkTimePump2
END_MACRO
#131 ND0502dosingError <= #120.out 1
#132 ND0502statRegimeP1M <= #120.out 2
#133 ND0502statRegimeP2M <= #120.out 3
#134 ND0502statRegimeByC <= #120.out 4
#135 ND0502statRegimeByWT <= #120.out 5
#136 DD1_AO3 <= #120.out 6
#137 DD10_AO0 <= #120.out 7
#138 ND0502counterP1 <= #120.out 8
#139 ND0502counterP2 <= #120.out 9
#140 ND0502workTimeP1 <= #120.out 10
#141 ND0502workTimeP2 <= #120.out 11
#142 DD4_DO.4 <= #120.out 12
#143 DD4_DO.5 <= #120.out 13
#144 AND(DD2_DO.1, DD5_DI.4)
#145 N0105statStartedP1 <= #144
#146 AND(DD5_DI.4, DD2_DO.2)
#147 N0105statStartedP2 <= #146
#148 MACRO Наполнение РЧВ02.03 (заслонка ЗДЭ02.25)(pin 1 "LS02.02раб.верх.уровень РЧВ": DD6_DI.14, pin 2 "LSA02.01 Перелив РЧВ": DD6_DI.13, pin 3 "статус ЗДЭ02.25 открыт": DD9_DI.0, pin 4 "статус ЗДЭ02.25 закрыт": DD9_DI.1, pin 5 "сброс аварий": alarmReset, pin 6 "время на открытие/закрытие": timeToOpenCloseValve)
	#149 OR(testZDE0225, pin 1)
	#150 NOT(pin 1)
	#151 ZDE0225:SimpleValve(inputOpen: #149, inputClose: #152, statusOpen: pin 3, statusClose: pin 4, reset: pin 5, timeToOpenClose: pin 6)
	out 1 "выход на открытие ЗДЭ02.25" <= #151.outputOpen
	#152 OR(#150, #153)
	out 2 "выход на закрытие ЗДЭ02.25" <= #151.outputClose
	out 3 "авария на открытие ЗДЭ02.25" <= #151.errorToOpen
	#153 NOT(pin 2)
	out 4 "авария на закрытие ЗДЭ02.25" <= #151.errorToClose
END_MACRO
#154 DD4_DO.0 <= #148.out 1
#155 DD4_DO.1 <= #148.out 2
#156 ZDE0225errorToOpen <= #148.out 3
#157 ZDE0225errorToClose <= #148.out 4
#158 MACRO управление Н02.04 (подача из РЧВ)(pin 1 "промывка ФС02.01/01": DD6_DI.20, pin 2 "промывка ФС02.01/02": DD6_DI.22, pin 3 "промывка ФС02.01/03": DD6_DI.24, pin 4 "промывка ФС02.01/04": DD6_DI.26, pin 5 "промывка ФС02.01/05": DD6_DI.28, pin 6 "промывка ФС02.01/06": DD6_DI.30, pin 7 "промывка ФС02.02/01": DD7_DI.0, pin 8 "промывка ФС02.02/02": DD7_DI.2, pin 9 "промывка ФС02.02/03": DD7_DI.4, pin 10 "промывка ФС02.02/04": DD7_DI.6, pin 11 "промывка ФС02.02/05": DD7_DI.8, pin 12 "промывка ФС02.02/06": DD7_DI.10, pin 13 "открыт КЭМ05.01": DD1_DI11, pin 14 "открыт КЭМ06.01": DD1_DI10, pin 15 "открыт КЭМ07.01": DD1_DI9, pin 16 "открыт КЭМ08.01": DD1_DI8, pin 17 "сухой ход Н02.04 (0=сух.ход)": DD5_DI.11, pin 18 "выбрать режим: Н02.04/01 - главный": N0204regimeP1M, pin 19 "выбрать режим: Н02.04/02 - главный": N0204regimeP2M, pin 20 "выбрать режим: по кол-ву включений": N0204regimeByC, pin 21 "выбрать режим: по наработке": N0204regimeWT, pin 22 "авария Н02.04/01 (0=авария)": DD5_DI.7, pin 23 "авария Н02.04/02 (0=авария)": DD5_DI.8, pin 24 "сброс аварий": alarmReset, pin 25 "сброс счетчика включений Н02.04/01": N0204resetCountP1, pin 26 "сброс счетчика включений Н02.04/02": N0204resetCountP2, pin 27 "сброс счетчика наработки Н02.04/01": N0204resetWorkTimeP1, pin 28 "сброс счетчика наработки Н02.04/02": N0204resetWorkTimeP2)
	(* Защита от сухого хода Н02.04 / (LS02.03) 0=сух.ход *)
	(* сброс самоподхвата реле *)
	(* Контроль открытия хотя бы одного из клапанов КЭМ *)
	(* Удержание сигнала на выключение насосов для / гарантированного сброса самоподхвата реле. *)
	(* Проверка, что фильтры 2 / ступени в регенерации (промывке) *)
	(* Проверка, что фильтры 1 / ступени в регенерации (промывке) *)
	#159 OR(pin 1, pin 2, pin 3, pin 4, pin 5, pin 6)
	#160 OR(#159, #161, #162)
	#161 OR(pin 7, pin 8, pin 9, pin 10, pin 11, pin 12)
	#162 OR(pin 13, pin 14, pin 15, pin 16)
	#163 N020401fTrigStop:F_TRIG(CLK: #170.pump1ON)
	#164 AND(#160, pin 17)
	#165 OR(#163.Q, #168.Q)
	#166 N0204stop:TOF(IN: #165, PT: T#1s)
	out 5 "стоп Н02.04" <= #166.Q
	#167 N0204chooseRegime:choosePumpRegime(start: #164, pump1Main: pin 18, pump2Main: pin 19, byCounter: #169, byWorkTime: pin 21)
	out 1 "выбран режим Н02.04/01 = главный" <= #167.pump1MainActive
	#168 N020402fTrigStop:F_TRIG(CLK: #170.pump2ON)
	out 2 "выбран режим Н02.04/02 = главный" <= #167.pump2MainActive
	out 3 "выбран режим по кол-ву включений" <= #167.byCounterActive
	#169 OR(pin 20, startInitializer)
	out 4 "выбран режим по наработке" <= #167.byWorkTimeActive
	#170 N0204manager:TwoPumpManager(startStopPump1: #167.startPump1, startStopPump2: #167.startPump2, alarmPump1: NOT pin 22, alarmPump2: NOT pin 23, alarmReset: pin 24, counterStart: #167.startByCounter, Pump1ResetCounter: pin 25, Pump2ResetCounter: pin 26, ValueToResetCounter: -, workTimeStart: #167.startByWorkTime, workTimePump1Reset: pin 27, workTimePump2Reset: pin 28)
	out 6 "пуск Н02.04/01" <= #170.pump1ON
	out 7 "пуск Н02.04/02" <= #170.pump2ON
	out 8 "счетчик включений Н02.04/01" <= #170.counterPump1
	out 9 "счетчик включений Н02.04/02" <= #170.counterPump2
	out 10 "счетчик наработки Н02.04/01" <= #170.currentWorkTimePump1
	out 11 "счетчик наработки Н02.04/02" <= #170.currentWorkTimePump2
END_MACRO
#171 N0204statRegimeP1M <= #158.out 1
#172 N0204statRegimeP2M <= #158.out 2
#173 N0204statRegimeByC <= #158.out 3
#174 N0204statRegimeWT <= #158.out 4
#175 DD4_DO.14 <= #158.out 5
#176 DD1_DO1 <= #158.out 6
#177 DD1_DO2 <= #158.out 7
#178 N0204counterP1 <= #158.out 8
#179 N0204counterP2 <= #158.out 9
#180 N0204workTimeP1 <= #158.out 10
#181 N0204workTimeP2 <= #158.out 11
#182 MACRO управление НД06.02 УПК(pin 1 "вход расходомера в куб/час": DD1_AI2_FT0102value, pin 2 "max производительность НД в мл/мин": ND0602setMaxDosVal, pin 3 "задание дозирования в мл/куб": ND0602setKoefProp, pin 4 "режим:1 насос главный": ND0602regimeP1M, pin 5 "режим: 2 насос главный": ND0602regimeP2M, pin 6 "режим: по наработке": ND0602regimeByWT, pin 7 "режим: по кол-ву включений": ND0602regimeByC, pin 8 "авария 1 насоса": DD6_DI.2, pin 9 "авария 2 насоса": DD6_DI.3, pin 10 "сброс аварий": alarmReset, pin 11 "сброс счетчика включений 1 насоса": ND0602resetCountP1, pin 12 "сброс ссчетчика включений 2 насоса": ND0602resetCountP2, pin 13 "сброс наработки 1 насоса": ND0602resetWorkTimeP1, pin 14 "сброс наработки 2 насоса": ND0602resetWorkTimeP2)
	(* Если на входе SEL = TRUE, / то нижнее значение, / иначе - то,что посередине. *)
	(* сигнал 4...20мА на НД06.02/01 *)
	(* сигнал 4...20мА на НД06.02/02 *)
	#183 SEL(#192.pump1ON, 4, #186.outputValue)
	#184 linTraf060201:LIN_TRAFO(IN: #183, IN_MIN: 4, IN_MAX: 20, OUT_MIN: 0, OUT_MAX: 1000)
	#185 REAL_TO_WORD(#184.OUT)
	out 6 "выход 4...20мА насоса 1" <= #185
	#186 ND0602dosing:DosingPumpProportional(flowValue: pin 1, setMinPumpDosingValue: -, setMaxPumpDosingValue: pin 2, minOutputValue: -, maxOutputValue: -, setKoeffProportionality: pin 3, minFlowToStart: -)
	out 1 "ошибка блока дозирования" <= #186.dosingError
	#187 SEL(#192.pump2ON, 4, #186.outputValue)
	#188 linTraf060202:LIN_TRAFO(IN: #187, IN_MIN: 4, IN_MAX: 20, OUT_MIN: 0, OUT_MAX: 1000)
	#189 REAL_TO_WORD(#188.OUT)
	out 7 "выход 4...20мА насоса 2" <= #189
	#190 ND0602regime:choosePumpRegime(start: #186.startDosingPump, pump1Main: pin 4, pump2Main: pin 5, byCounter: #191, byWorkTime: pin 6)
	out 2 "статус: 1 насос главный" <= #190.pump1MainActive
	out 3 "статус: 2 насос главный" <= #190.pump2MainActive
	out 4 "статус: по кол-ву включений" <= #190.byCounterActive
	#191 OR(pin 7, startInitializer)
	out 5 "статус: по наработке" <= #190.byWorkTimeActive
	#192 ND0602manager:TwoPumpManager(startStopPump1: #190.startPump1, startStopPump2: #190.startPump2, alarmPump1: #193, alarmPump2: #194, alarmReset: pin 10, counterStart: #190.startByCounter, Pump1ResetCounter: pin 11, Pump2ResetCounter: pin 12, ValueToResetCounter: -, workTimeStart: #190.startByWorkTime, workTimePump1Reset: pin 13, workTimePump2Reset: pin 14)
	out 12 "сигнал на включение насоса 1" <= #192.pump1ON
	#193 NOT(pin 8)
	out 13 "сигнал на включение насоса 2" <= #192.pump2ON
	out 8 "счетчик включений насоса 1" <= #192.counterPump1
	#194 NOT(pin 9)
	out 9 "счетчик включений насоса 2" <= #192.counterPump2
	out 10 "счетчик наработки насоса 1" <= #192.currentWorkTimePump1
	out 11 "счетчик наработки насоса 2" <= #192.currentWorkTimePump2
END_MACRO
#195 ND0602dosingError <= #182.out 1
#196 ND0602statRegimeP1M <= #182.out 2
#197 ND0602statRegimeP2M <= #182.out 3
#198 ND0602statRegimeByC <= #182.out 4
#199 ND0602statRegimeByWT <= #182.out 5
#200 DD10_AO1 <= #182.out 6
#201 DD10_AO2 <= #182.out 7
#202 ND0602counterP1 <= #182.out 8
#203 ND0602counterP2 <= #182.out 9
#204 ND0602workTimeP1 <= #182.out 10
#205 ND0602workTimeP2 <= #182.out 11
#206 DD4_DO.6 <= #182.out 12
#207 DD4_DO.7 <= #182.out 13
#208 OR(errorToOpenZDE0301, errorToCloseZDE0301, errorToOpenZDE0302, errorToCloseZDE0302)
#209 OR(DD5_DI.27, #208)
#210 OR(#208, DD5_DI.29)
#211 MACRO Работа УФО03.01(pin 1 "Работа УФО03.01/01": statusUFO030101started, pin 2 "Работа УФО03.01/02": statusUFO030102started, pin 3 "Значение расхода от FT01.02": DD1_AI2_FT0102value, pin 4 "мин.допустимый расход для насосов Н01.05": N0105minFlow, pin 5 "Задержка включения УФО на создание потока": UFO0301startDelayTime, pin 6 "выбор режим: УФО03.01/01 главное": UFO0301regimeP1M, pin 7 "выбор режим: УФО03.01/02 главное": UFO0301regimeP2M, pin 8 "выбор режим: по кол-ву включений": UFO0301regimeByC, pin 9 "выбор режим: по наработке": UFO0301regimeWT, pin 10 "авария УФО03.01/01": #209, pin 11 "авария УФО03.01/02": #210, pin 12 "сброс аварий": alarmReset, pin 13 "сброс счетчика включений УФО03.01/01": UFO0301resetCountP1, pin 14 "сброс счетчика включений УФО03.01/02": UFO0301resetCountP2, pin 15 "сброс счетчика наработки УФО03.01/01": UFO0301resetWorkTimeP1, pin 16 "сброс счетчика наработки УФО03.01/02": UFO0301resetWorkTimeP2)
	(* Включаем УФО, если расходомер показывает расход больше, / чем заданный как минимально допустимый для работы насосов Н01.05. *)
	(* Задержка старта УФО *)
	(* Для подачи предостережения на пульте / оператора (при необходимости), а также / сигнализации лампой АВАРИЯ. *)
	(* Контроль, если УФО включили вручную, / а потока при этом нет. *)
	#212 OR(pin 1, pin 2)
	#213 AND(#212, #214)
	out 1 "УФО вкл без потока" <= #213
	#214 NOT(#216.Q)
	#215 GE(pin 3, pin 4)
	#216 UFO0301startDelay:TON(IN: #215, PT: pin 5)
	#217 UFO0301regimeManager:choosePumpRegime(start: #216.Q, pump1Main: pin 6, pump2Main: pin 7, byCounter: #218, byWorkTime: pin 9)
	out 2 "активен режим - главное УФО 03.01/01" <= #217.pump1MainActive
	out 3 "активен режим - главное УФО 03.01/02" <= #217.pump2MainActive
	out 4 "активен режим - по кол-ву включений" <= #217.byCounterActive
	#218 OR(startInitializer, pin 8)
	out 5 "активен режим - по наработке" <= #217.byWorkTimeActive
	#219 UFO0301manager:TwoPumpManager(startStopPump1: #217.startPump1, startStopPump2: #217.startPump2, alarmPump1: pin 10, alarmPump2: pin 11, alarmReset: pin 12, counterStart: #217.startByCounter, Pump1ResetCounter: pin 13, Pump2ResetCounter: pin 14, ValueToResetCounter: -, workTimeStart: #217.startByWorkTime, workTimePump1Reset: pin 15, workTimePump2Reset: pin 16)
	out 6 "авт. пуск УФО03.01/01" <= #219.pump1ON
	out 7 "авт. пуск УФО03.01/02" <= #219.pump2ON
	out 8 "счетчик включений УФО03.01/01" <= #219.counterPump1
	out 9 "счетчик включений УФО03.01/02" <= #219.counterPump2
	out 10 "счетчик наработки УФО03.01/01" <= #219.currentWorkTimePump1
	out 11 "счетчик наработки УФО03.01/02" <= #219.currentWorkTimePump2
END_MACRO
#220 UFO0301noFlowAttention <= #211.out 1
#221 UFO0301statRegimeP1M <= #211.out 2
#222 UFO0301statRegimeP2M <= #211.out 3
#223 UFO0301statRegimeByC <= #211.out 4
#224 UFO0301statRegimeWT <= #211.out 5
#225 UFO0301counterP1 <= #211.out 8
#226 UFO0301counterP2 <= #211.out 9
#227 UFO0301workTimeP1 <= #211.out 10
#228 UFO0301workTimeP2 <= #211.out 11
#229 MACRO работа задвижек перед УФО и автом.пуск(pin 1 "сигнал на пуск УФО03.01/01": #211.out 6, pin 2 "сигнал на пуск УФО03.01/02": #211.out 7)
	(* 1 = открыть ЗДЭ03.02 / 0 = закрыть ЗДЭ03.02 *)
	(* 1 = открыть ЗДЭ03.01 / 0 = закрыть ЗДЭ03.01 *)
	(* 1 = тест задвижек ЗДЭ / 0 = возможность автом.пуска УФО *)
	(* авт.пускУФО03.01/01 *)
	(* авт.пускУФО03.01/02 *)
	(* авт.стопУФО03.01/01 *)
	(* авт.стопУФО03.01/02 *)
	#230 NOT(testZDE03)
	#231 NOT(testZDE03)
	#232 UFO030101startTrig:R_TRIG(CLK: #234)
	#233 UFO030101start <= #232.Q
	#234 AND(#230, #237, DD1_DI12)
	#235 UFO030101stopTrig:F_TRIG(CLK: #234)
	#236 UFO030101stop <= #235.Q
	#237 SEL(testZDE03, pin 1, manualZDE0301)
	#238 ZDE0301:SimpleValve(inputOpen: #237, inputClose: NOT #237, statusOpen: DD1_DI12, statusClose: DD1_DI13, reset: alarmReset, timeToOpenClose: timeToOpenCloseValve)
	#239 DD4_DO.16 <= #238.outputOpen
	#240 DD4_DO.17 <= #238.outputClose
	#241 errorToOpenZDE0301 <= #238.errorToOpen
	#242 errorToCloseZDE0301 <= #238.errorToClose
	#243 UFO030102startTrig:R_TRIG(CLK: #245)
	#244 UFO030102start <= #243.Q
	#245 AND(#231, #248, DD1_DI14)
	#246 UFO030102stopTrig:F_TRIG(CLK: #245)
	#247 UFO030102stop <= #246.Q
	#248 SEL(testZDE03, pin 2, manualZDE0302)
	#249 ZDE0302:SimpleValve(inputOpen: #248, inputClose: NOT #248, statusOpen: DD1_DI14, statusClose: DD1_DI15, reset: alarmReset, timeToOpenClose: timeToOpenCloseValve)
	#250 DD4_DO.18 <= #249.outputOpen
	#251 DD4_DO.19 <= #249.outputClose
	#252 errorToOpenZDE0302 <= #249.errorToOpen
	#253 errorToCloseZDE0302 <= #249.errorToClose
END_MACRO
#254 MACRO управление НД06.03 УПК(pin 1 "вход расходомера в куб/час": DD1_AI1_FT0101value, pin 2 "max производительность НД в мл/мин": ND0603setMaxDosVal, pin 3 "задание дозирования в мл/куб": ND0603setKoefProp, pin 4 "режим:1 насос главный": ND0603regimeP1M, pin 5 "режим: 2 насос главный": ND0603regimeP2M, pin 6 "режим: по наработке": ND0603regimeByWT, pin 7 "режим: по кол-ву включений": ND0603regimeByC, pin 8 "авария 1 насоса": DD6_DI.4, pin 9 "авария 2 насоса": DD6_DI.5, pin 10 "сброс аварий": alarmReset, pin 11 "сброс счетчика включений 1 насоса": ND0603resetCountP1, pin 12 "сброс ссчетчика включений 2 насоса": ND0603resetCountP2, pin 13 "сброс наработки 1 насоса": ND0603resetWorkTimeP1, pin 14 "сброс наработки 2 насоса": ND0603resetWorkTimeP2)
	(* Если на входе SEL = TRUE, / то нижнее значение, / иначе - то,что посередине. *)
	(* сигнал 4...20мА на НД06.03/01 *)
	(* сигнал 4...20мА на НД06.03/02 *)
	#255 SEL(#264.pump1ON, 4, #258.outputValue)
	#256 linTraf060301:LIN_TRAFO(IN: #255, IN_MIN: 4, IN_MAX: 20, OUT_MIN: 0, OUT_MAX: 1000)
	#257 REAL_TO_WORD(#256.OUT)
	out 6 "выход 4...20мА насоса 1" <= #257
	#258 ND0603dosing:DosingPumpProportional(flowValue: pin 1, setMinPumpDosingValue: -, setMaxPumpDosingValue: pin 2, minOutputValue: -, maxOutputValue: -, setKoeffProportionality: pin 3, minFlowToStart: -)
	out 1 "ошибка блока дозирования" <= #258.dosingError
	#259 SEL(#264.pump2ON, 4, #258.outputValue)
	#260 linTraf060302:LIN_TRAFO(IN: #259, IN_MIN: 4, IN_MAX: 20, OUT_MIN: 0, OUT_MAX: 1000)
	#261 REAL_TO_WORD(#260.OUT)
	out 7 "выход 4...20мА насоса 2" <= #261
	#262 ND0603regime:choosePumpRegime(start: #258.startDosingPump, pump1Main: pin 4, pump2Main: pin 5, byCounter: #263, byWorkTime: pin 6)
	out 2 "статус: 1 насос главный" <= #262.pump1MainActive
	out 3 "статус: 2 насос главный" <= #262.pump2MainActive
	out 4 "статус: по кол-ву включений" <= #262.byCounterActive
	#263 OR(pin 7, startInitializer)
	out 5 "статус: по наработке" <= #262.byWorkTimeActive
	#264 ND0603manager:TwoPumpManager(startStopPump1: #262.startPump1, startStopPump2: #262.startPump2, alarmPump1: #265, alarmPump2: #266, alarmReset: pin 10, counterStart: #262.startByCounter, Pump1ResetCounter: pin 11, Pump2ResetCounter: pin 12, ValueToResetCounter: -, workTimeStart: #262.startByWorkTime, workTimePump1Reset: pin 13, workTimePump2Reset: pin 14)
	out 12 "сигнал на включение насоса 1" <= #264.pump1ON
	#265 NOT(pin 8)
	out 13 "сигнал на включение насоса 2" <= #264.pump2ON
	out 8 "счетчик включений насоса 1" <= #264.counterPump1
	#266 NOT(pin 9)
	out 9 "счетчик включений насоса 2" <= #264.counterPump2
	out 10 "счетчик наработки насоса 1" <= #264.currentWorkTimePump1
	out 11 "счетчик наработки насоса 2" <= #264.currentWorkTimePump2
END_MACRO
#267 ND0603dosingError <= #254.out 1
#268 ND0603statRegimeP1M <= #254.out 2
#269 ND0603statRegimeP2M <= #254.out 3
#270 ND0603statRegimeByC <= #254.out 4
#271 ND0603statRegimeByWT <= #254.out 5
#272 DD10_AO3 <= #254.out 6
#273 DD10_AO4 <= #254.out 7
#274 ND0603counterP1 <= #254.out 8
#275 ND0603counterP2 <= #254.out 9
#276 ND0603workTimeP1 <= #254.out 10
#277 ND0603workTimeP2 <= #254.out 11
#278 DD4_DO.8 <= #254.out 12
#279 DD4_DO.9 <= #254.out 13
#280 MACRO управление Н04.04 (дренажные)(pin 1 "защита от сухого хода Н04.04": DD5_DI.18, pin 2 "автоматич.пускН04.04": DD5_DI.19, pin 3 "режим Н04.04/01 главный": N0404regimeP1M, pin 4 "режим Н04.04/02 главный": N0404regimeP2M, pin 5 "режим по кол-ву включений": N0404regimeByC, pin 6 "режим по наработке": N0404regimeWT, pin 7 "авария Н04.04/01": DD5_DI.15, pin 8 "авария Н04.04/02": DD5_DI.14, pin 9 "сброс аварий": alarmReset, pin 10 "сброс счетчика включений Н04.04/01": N0404resetCountP1, pin 11 "сброс счетчика включений Н04.04/02": N0404resetCountP2, pin 12 "сброс счетчика наработки Н04.04/01": N0404resetWorkTimeP1, pin 13 "сброс счетчика наработки Н04.04/02": N0404resetWorkTimeP2)
	(* 0=авария *)
	(* сухой ход Н04.04 / 0=защита *)
	(* от поплавка *)
	(* насосы имеют электрическую блокировку / от одновременного включения *)
	(* Излишняя перестраховка по сухому ходу, / на уровне реле уже все отрабатывается. *)
	(* сбрасывает самоподхват пускового реле *)
	#281 NOT(pin 1)
	out 1 "стоп Н04.04" <= #281
	#282 AND(pin 1, pin 2)
	#283 N0401choosePumpRegime:choosePumpRegime(start: #282, pump1Main: pin 3, pump2Main: pin 4, byCounter: #284, byWorkTime: pin 6)
	out 2 "выбран режим: Н04.04/01 главный" <= #283.pump1MainActive
	out 3 "выбран режим: Н04.04/02 главный" <= #283.pump2MainActive
	out 4 "выбран режим: по кол-ву включений" <= #283.byCounterActive
	#284 OR(startInitializer, pin 5)
	out 5 "выбран режим: по наработке" <= #283.byWorkTimeActive
	#285 N0404twoPumpManager:TwoPumpManager(startStopPump1: #283.startPump1, startStopPump2: #283.startPump2, alarmPump1: #286, alarmPump2: #287, alarmReset: pin 9, counterStart: #283.startByCounter, Pump1ResetCounter: pin 10, Pump2ResetCounter: pin 11, ValueToResetCounter: -, workTimeStart: #283.startByWorkTime, workTimePump1Reset: pin 12, workTimePump2Reset: pin 13)
	out 6 "пуск Н04.04/01" <= #285.pump1ON
	#286 NOT(pin 7)
	out 7 "пуск Н04.04/02" <= #285.pump2ON
	out 8 "счетчик кол-ва включений Н04.04/01" <= #285.counterPump1
	#287 NOT(pin 8)
	out 9 "счетчик кол-ва включений Н04.04/02" <= #285.counterPump2
	out 10 "счетчик времени наработки Н04.04/01" <= #285.currentWorkTimePump1
	out 11 "счетчик времени наработки Н04.04/02" <= #285.currentWorkTimePump2
END_MACRO
#288 DD4_DO.15 <= #280.out 1
#289 N0404statRegimeP1M <= #280.out 2
#290 N0404statRegimeP2M <= #280.out 3
#291 N0404statRegimeByC <= #280.out 4
#292 N0404statRegimeWT <= #280.out 5
#293 DD1_DO5 <= #280.out 6
#294 DD1_DO6 <= #280.out 7
#295 N0404counterP1 <= #280.out 8
#296 N0404counterP2 <= #280.out 9
#297 N0404workTimeP1 <= #280.out 10
#298 N0404workTimeP2 <= #280.out 11
#299 MACRO управление НД07.03 УПЩ (поддержка рН, ПИД-регулятор)(pin 1 "вход рН-метра QE01.01": DD1_AI3_QE0101value, pin 2 "уставка рН": ND0703pHsetValue, pin 3 "режим:1 насос главный": ND0703regimeP1M, pin 4 "режим: 2 насос главный": ND0703regimeP2M, pin 5 "режим: по наработке": ND0703regimeByWT, pin 6 "режим: по кол-ву включений": ND0703regimeByC, pin 7 "авария 1 насоса": DD6_DI.6, pin 8 "авария 2 насоса": DD6_DI.7, pin 9 "сброс аварий": alarmReset, pin 10 "сброс счетчика включений 1 насоса": ND0703resetCountP1, pin 11 "сброс счетчика включений 2 насоса": ND0703resetCountP2, pin 12 "сброс наработки 1 насоса": ND0703resetWorkTimeP1, pin 13 "сброс наработки 2 насоса": ND0703resetWorkTimeP2, pin 14 "ручное управл.выходом Y (4...20мА)": ND0703YoutManual, pin 15 "1=ручное/0=автомат.управл.": ND0703YmanAuto, pin 16 "вход расходомера FT01.01 (куб.м/час)": DD1_AI1_FT0101value, pin 17 "коэфф.I": ND0703koeffI, pin 18 "коэфф.D": ND0703koeffD, pin 19 "коэфф.Р": ND0703koeffP)
	(* min расход в кубометрах в час / для неачала дозирования. *)
	(* Если на входе SEL = TRUE, / то нижнее значение, / иначе - то,что посередине. *)
	(* сигнал 4...20мА на НД07.03/01 *)
	(* сигнал 4...20мА на НД07.03/02 *)
	#300 ND0703pidReg:PID(ACTUAL: pin 1, SET_POINT: pin 2, KP: pin 19, TN: pin 17, TV: pin 18, Y_MANUAL: pin 14, Y_OFFSET: 12, Y_MIN: 0, Y_MAX: 1000, MANUAL: pin 15, RESET: #300.OVERFLOW)
	#301 SEL(#308.pump1ON, 0, #300.Y)
	#302 REAL_TO_WORD(#301)
	out 5 "выход 4...20мА насоса 1" <= #302
	#303 SEL(#308.pump2ON, 0, #300.Y)
	#304 REAL_TO_WORD(#303)
	out 6 "выход 4...20мА насоса 2" <= #304
	#305 GE(pin 16, 10)
	#306 ND0703regime:choosePumpRegime(start: #305, pump1Main: pin 3, pump2Main: pin 4, byCounter: #307, byWorkTime: pin 5)
	out 1 "статус: 1 насос главный" <= #306.pump1MainActive
	out 2 "статус: 2 насос главный" <= #306.pump2MainActive
	out 3 "статус: по кол-ву включений" <= #306.byCounterActive
	out 4 "статус: по наработке" <= #306.byWorkTimeActive
	#307 OR(pin 6, startInitializer)
	#308 ND0703manager:TwoPumpManager(startStopPump1: #306.startPump1, startStopPump2: #306.startPump2, alarmPump1: #309, alarmPump2: #310, alarmReset: pin 9, counterStart: #306.startByCounter, Pump1ResetCounter: pin 10, Pump2ResetCounter: pin 11, ValueToResetCounter: -, workTimeStart: #306.startByWorkTime, workTimePump1Reset: pin 12, workTimePump2Reset: pin 13)
	out 11 "сигнал на включение насоса 1" <= #308.pump1ON
	#309 NOT(pin 7)
	out 12 "сигнал на включение насоса 2" <= #308.pump2ON
	out 7 "счетчик включений насоса 1" <= #308.counterPump1
	#310 NOT(pin 8)
	out 8 "счетчик включений насоса 2" <= #308.counterPump2
	out 9 "счетчик наработки насоса 1" <= #308.currentWorkTimePump1
	out 10 "счетчик наработки насоса 2" <= #308.currentWorkTimePump2
END_MACRO
#311 ND0703statRegimeP1M <= #299.out 1
#312 ND0703statRegimeP2M <= #299.out 2
#313 ND0703statRegimeByC <= #299.out 3
#314 ND0703statRegimeByWT <= #299.out 4
#315 DD10_AO5 <= #299.out 5
#316 DD10_AO6 <= #299.out 6
#317 ND0703counterP1 <= #299.out 7
#318 ND0703counterP2 <= #299.out 8
#319 ND0703workTimeP1 <= #299.out 9
#320 ND0703workTimeP2 <= #299.out 10
#321 DD4_DO.10 <= #299.out 11
#322 DD4_DO.11 <= #299.out 12
#323 MACRO импульсный счетчик FQS0301(pin 1 "вход от счетчика": DD6_DI.19, pin 2 "вес импульса счетчика": FQS0301impulsValue, pin 3 "сброс счетчика": FQS0301reset, pin 4 "величина коррекции счетчика": FQS0301correction, pin 5 "прибавить коррекцию": FQS0301addCorrection, pin 6 "вычесть коррекцию": FQS0301deleteCorrection)
	(* число, коорое будем прибавлять или / вычитать из накопленной суммы стоков. *)
	(* коррекция показаний счетчика. *)
	(* Если в результате коррекции накопленная сумма станет меньше нуля, то она принудительно станет равна нулю. *)
	(* значение в REAL (в какой-то момент начинает / отображаться в экспоненциальной форме) *)
	(* сброс показаний счетчика *)
	#324 FQS0301rTrig:R_TRIG(CLK: pin 1)
	#325 ADD(EN: #324.Q, FQS0301totalAmount, pin 2)
	out 1 "накопленная сумма стоков (REAL)" <= #325
	#326 FQS0301resetRtrig:R_TRIG(CLK: pin 3)
	#327 MOVE(EN: #326.Q, 0)
	#328 FQS0301totalAmount <= #327
	#329 FQS0301addCorrRtrig:R_TRIG(CLK: pin 5)
	#330 ADD(EN: #329.Q, FQS0301totalAmount, pin 4)
	#331 FQS0301totalAmount <= #330
	#332 FQS0301deleteCorrRtrig:R_TRIG(CLK: pin 6)
	#333 SUB(EN: #332.Q, FQS0301totalAmount, pin 4)
	#334 FQS0301totalAmount <= #333
	#335 LT(FQS0301totalAmount, 0)
	#336 MOVE(EN: #335, 0)
	#337 FQS0301totalAmount <= #336
END_MACRO
#338 FQS0301totalAmount <= #323.out 1
#339 MACRO управление НД08.03 УПФ(pin 1 "вход расходомера в куб/час": DD1_AI1_FT0101value, pin 2 "max производительность НД в мл/мин": ND0803setMaxDosVal, pin 3 "задание дозирования в мл/куб": ND0803setKoefProp, pin 4 "режим:1 насос главный": ND0803regimeP1M, pin 5 "режим: 2 насос главный": ND0803regimeP2M, pin 6 "режим: по наработке": ND0803regimeByWT, pin 7 "режим: по кол-ву включений": ND0803regimeByC, pin 8 "авария 1 насоса": DD5_DI.12, pin 9 "авария 2 насоса": DD5_DI.13, pin 10 "сброс аварий": alarmReset, pin 11 "сброс счетчика включений 1 насоса": ND0803resetCountP1, pin 12 "сброс ссчетчика включений 2 насоса": ND0803resetCountP2, pin 13 "сброс наработки 1 насоса": ND0803resetWorkTimeP1, pin 14 "сброс наработки 2 насоса": ND0803resetWorkTimeP2, pin 15 "сухой ход 1 насоса": DD1_DI6, pin 16 "сухой ход 2 насоса": DD1_DI7)
	(* Если на входе SEL = TRUE, / то нижнее значение, / иначе - то,что посередине. *)
	(* сигнал 4...20мА на НД08.03/01 *)
	(* сигнал 4...20мА на НД08.03/02 *)
	#340 SEL(#349.pump1ON, 0, #341.outputValue)
	out 6 "выход 4...20мА насоса 1" <= #340
	#341 ND0803dosing:DosingPumpProportional(flowValue: pin 1, setMinPumpDosingValue: -, setMaxPumpDosingValue: pin 2, minOutputValue: -, maxOutputValue: -, setKoeffProportionality: pin 3, minFlowToStart: -)
	out 1 "ошибка блока дозирования" <= #341.dosingError
	#342 SEL(#349.pump2ON, 0, #341.outputValue)
	out 7 "выход 4...20мА насоса 2" <= #342
	#343 ND0803regime:choosePumpRegime(start: #341.startDosingPump, pump1Main: pin 4, pump2Main: pin 5, byCounter: #344, byWorkTime: pin 6)
	out 2 "статус: 1 насос главный" <= #343.pump1MainActive
	out 3 "статус: 2 насос главный" <= #343.pump2MainActive
	out 4 "статус: по кол-ву включений" <= #343.byCounterActive
	#344 OR(pin 7, startInitializer)
	out 5 "статус: по наработке" <= #343.byWorkTimeActive
	out 12 "сигнал на включение насоса 1" <= #349.pump1ON
	#345 NOT(pin 8)
	#346 OR(#345, pin 15)
	out 13 "сигнал на включение насоса 2" <= #349.pump2ON
	#347 NOT(pin 9)
	#348 OR(#347, pin 16)
	#349 ND0803manager:TwoPumpManager(startStopPump1: #343.startPump1, startStopPump2: #343.startPump2, alarmPump1: #346, alarmPump2: #348, alarmReset: pin 10, counterStart: #343.startByCounter, Pump1ResetCounter: pin 11, Pump2ResetCounter: pin 12, ValueToResetCounter: -, workTimeStart: #343.startByWorkTime, workTimePump1Reset: pin 13, workTimePump2Reset: pin 14)
	out 8 "счетчик включений насоса 1" <= #349.counterPump1
	out 9 "счетчик включений насоса 2" <= #349.counterPump2
	out 10 "счетчик наработки насоса 1" <= #349.currentWorkTimePump1
	out 11 "счетчик наработки насоса 2" <= #349.currentWorkTimePump2
END_MACRO
#350 ND0803dosingError <= #339.out 1
#351 ND0803statRegimeP1M <= #339.out 2
#352 ND0803statRegimeP2M <= #339.out 3
#353 ND0803statRegimeByC <= #339.out 4
#354 ND0803statRegimeByWT <= #339.out 5
#355 DD1_AO1 <= #339.out 6
#356 DD1_AO2 <= #339.out 7
#357 ND0803counterP1 <= #339.out 8
#358 ND0803counterP2 <= #339.out 9
#359 ND0803workTimeP1 <= #339.out 10
#360 ND0803workTimeP2 <= #339.out 11
#361 DD1_DO3 <= #339.out 12
#362 DD1_DO4 <= #339.out 13
#363 AND(DD1_DI5, DD1_DI4, DD6_DI.11)
#364 DD1_DO8 <= #363
#365 EQ(lastError, 0)
#366 alarmPLKnetworkDelay:TOF(IN: #365, PT: T#20s)
#367 NOT(#366.Q)
#368 alarmPLKnetwork <= #367
#369 MACRO управление НД08.04 УПФ(pin 1 "насос Н04.01 работает": DD7_DI.13, pin 2 "авария НД08.04": DD6_DI.16, pin 3 "уставкаНД08.04(0...100%)": ND0804doseValue)
	(* Преобразует сигнал 0...100 / пропорционально в 4...20мА *)
	#370 AND(pin 1, pin 2)
	out 1 "пуск/стоп НД08.04" <= #370
	#371 ND0804linearTransformator:LIN_TRAFO(IN: pin 3, IN_MIN: 0, IN_MAX: 100, OUT_MIN: 0, OUT_MAX: 1000)
	#372 REAL_TO_WORD(#371.OUT)
	out 2 "управление НД08.04 (4...20мА)" <= #372
	out 3 "ошибка блока дозирования" <= #371.ERROR
END_MACRO
#373 DD4_DO.12 <= #369.out 1
#374 DD10_AO7 <= #369.out 2
#375 ND0804dosingError <= #369.out 3
#376 NOT(DD6_DI.0)
#377 alarmND050201 <= #376
#378 NOT(DD6_DI.23)
#379 alarmFS020102 <= #378
#380 NOT(DD9_DI.14)
#381 alarmZDE0211power <= #380
#382 NOT(DD6_DI.1)
#383 alarmND050202 <= #382
#384 NOT(DD6_DI.25)
#385 alarmFS020103 <= #384
#386 NOT(DD9_DI.15)
#387 alarmZDE0212power <= #386
#388 NOT(DD6_DI.2)
#389 alarmND060201 <= #388
#390 NOT(DD6_DI.27)
#391 alarmFS020104 <= #390
#392 NOT(DD9_DI.16)
#393 alarmZDE0213power <= #392
#394 NOT(DD6_DI.3)
#395 alarmND060202 <= #394
#396 NOT(DD6_DI.29)
#397 alarmFS020105 <= #396
#398 NOT(DD9_DI.17)
#399 alarmZDE0214power <= #398
#400 MACRO контроль включения мешалок(pin 1 "работа НД06.02/01": DD4_DO.6, pin 2 "работа НД06.02/02": DD4_DO.7, pin 3 "работа НД06.03/01": DD4_DO.8, pin 4 "работа НД06.03/02": DD4_DO.9, pin 5 "работа мешалки М06.04": DD5_DI.21, pin 6 "работа НД07.03/01": DD4_DO.10, pin 7 "работа НД07.03/02": DD4_DO.11, pin 8 "работа мешалки М07.02": DD5_DI.23, pin 9 "работа НД08.03/01": DD1_DO3, pin 10 "работа НД08.03/02": DD1_DO4, pin 11 "работа НД08.04": DD4_DO.12, pin 12 "работа мешалки М08.02": DD5_DI.25)
	#401 OR(pin 1, pin 2, pin 3, pin 4)
	#402 AND(#401, #403)
	out 1 "дозирования при выключенной М06.04" <= #402
	#403 NOT(pin 5)
	#404 OR(pin 6, pin 7)
	#405 AND(#404, #406)
	out 2 "дозирования при выключенной М07.02" <= #405
	#406 NOT(pin 8)
	#407 OR(pin 9, pin 10, pin 11)
	#408 AND(#407, #409)
	out 3 "дозирования при выключенной М08.02" <= #408
	#409 NOT(pin 12)
END_MACRO
#410 M0604attention <= #400.out 1
#411 M0702attention <= #400.out 2
#412 M0802attention <= #400.out 3
#413 NOT(DD6_DI.4)
#414 alarmND060301 <= #413
#415 NOT(DD6_DI.31)
#416 alarmFS020106 <= #415
#417 NOT(DD9_DI.18)
#418 alarmZDE0215power <= #417
#419 NOT(DD6_DI.5)
#420 alarmND060302 <= #419
#421 NOT(DD7_DI.1)
#422 alarmFS020201 <= #421
#423 NOT(DD9_DI.19)
#424 alarmZDE0216power <= #423
#425 NOT(DD6_DI.6)
#426 alarmND070301 <= #425
#427 NOT(DD7_DI.3)
#428 alarmFS020202 <= #427
#429 NOT(DD9_DI.20)
#430 alarmZDE0217power <= #429
#431 NOT(DD6_DI.7)
#432 alarmND070302 <= #431
#433 NOT(DD7_DI.5)
#434 alarmFS020203 <= #433
#435 NOT(DD9_DI.21)
#436 alarmZDE0218power <= #435
#437 NOT(DD5_DI.12)
#438 alarmND080301 <= #437
#439 NOT(DD7_DI.7)
#440 alarmFS020204 <= #439
#441 NOT(DD9_DI.22)
#442 alarmZDE0219power <= #441
#443 NOT(DD5_DI.13)
#444 alarmND080302 <= #443
#445 NOT(DD7_DI.9)
#446 alarmFS020205 <= #445
#447 NOT(DD9_DI.23)
#448 alarmZDE0220power <= #447
#449 NOT(DD6_DI.16)
#450 alarmND0804 <= #449
#451 NOT(DD7_DI.11)
#452 alarmFS020206 <= #451
#453 NOT(DD9_DI.24)
#454 alarmZDE0221power <= #453
#455 NOT(DD6_DI.11)
#456 alarmOGM0104overload <= #455
#457 NOT(DD9_DI.4)
#458 alarmZDE0201power <= #457
#459 NOT(DD9_DI.25)
#460 alarmZDE0222power <= #459
#461 MACRO переменные для обмена с панелью()
	#462 MACRO PSW регистры на передачу в панель (отображение)()
		(* panFQS0301totalAmount - переменная отображена сразу на выходе соответствующего макроса (учет очищенных стоков). / Здесь не хранится. *)
		(* PSW регистры на передачу в панель (отображение) *)
		#463 panFT0101value <= DD1_AI1_FT0101value
		#464 panQE0101value <= DD1_AI3_QE0101value
		#465 panFT0102value <= DD1_AI2_FT0102value
		#466 panQE0102value <= DD1_AI4_QE0102value
		#467 panFPKpressureValue <= DD1_AI5_FPKpressureValue
		#468 panFQS0301total <= FQS0301totalAmount
		#469 panTemperature <= temperatureValue
		#470 MACRO Время наработки и кол-во включений агрегатов()
			#471 workTimeND050201:TimeFromWorkTime(input: ND0502workTimeP1)
			#472 panND050201workDays <= #471.days
			#473 panND050201workHours <= #471.hours
			#474 panND050201workMinutes <= #471.minutes
			#475 panND050201workSeconds <= #471.seconds
			#476 workTimeND050202:TimeFromWorkTime(input: ND0502workTimeP2)
			#477 panND050202workDays <= #476.days
			#478 panND050202workHours <= #476.hours
			#479 panND050202workMinutes <= #476.minutes
			#480 panND050202workSeconds <= #476.seconds
			#481 panND0502counterP1 <= ND0502counterP1
			#482 panND0502counterP2 <= ND0502counterP2
			#483 workTimeND060201:TimeFromWorkTime(input: ND0602workTimeP1)
			#484 panND060201workDays <= #483.days
			#485 panND060201workHours <= #483.hours
			#486 panND060201workMinutes <= #483.minutes
			#487 panND060201workSeconds <= #483.seconds
			#488 workTimeND060202:TimeFromWorkTime(input: ND0602workTimeP2)
			#489 panND060202workDays <= #488.days
			#490 panND060202workHours <= #488.hours
			#491 panND060202workMinutes <= #488.minutes
			#492 panND060202workSeconds <= #488.seconds
			#493 panND0602counterP1 <= ND0602counterP1
			#494 panND0602counterP2 <= ND0602counterP2
			#495 workTimeND060301:TimeFromWorkTime(input: ND0603workTimeP1)
			#496 panND060301workDays <= #495.days
			#497 panND060301workHours <= #495.hours
			#498 panND060301workMinutes <= #495.minutes
			#499 panND060301workSeconds <= #495.seconds
			#500 workTimeND060302:TimeFromWorkTime(input: ND0603workTimeP2)
			#501 panND060302workDays <= #500.days
			#502 panND060302workHours <= #500.hours
			#503 panND060302workMinutes <= #500.minutes
			#504 panND060302workSeconds <= #500.seconds
			#505 panND0603counterP1 <= ND0603counterP1
			#506 panND0603counterP2 <= ND0603counterP2
			#507 workTimeND070301:TimeFromWorkTime(input: ND0703workTimeP1)
			#508 panND070301workDays <= #507.days
			#509 panND070301workHours <= #507.hours
			#510 panND070301workMinutes <= #507.minutes
			#511 panND070301workSeconds <= #507.seconds
			#512 workTimeND070302:TimeFromWorkTime(input: ND0703workTimeP2)
			#513 panND070302workDays <= #512.days
			#514 panND070302workHours <= #512.hours
			#515 panND070302workMinutes <= #512.minutes
			#516 panND070302workSeconds <= #512.seconds
			#517 panND0703counterP1 <= ND0703counterP1
			#518 panND0703counterP2 <= ND0703counterP2
			#519 workTimeND080301:TimeFromWorkTime(input: ND0803workTimeP1)
			#520 panND080301workDays <= #519.days
			#521 panND080301workHours <= #519.hours
			#522 panND080301workMinutes <= #519.minutes
			#523 panND080301workSeconds <= #519.seconds
			#524 workTimeND080302:TimeFromWorkTime(input: ND0803workTimeP2)
			#525 panND080302workDays <= #524.days
			#526 panND080302workHours <= #524.hours
			#527 panND080302workMinutes <= #524.minutes
			#528 panND080302workSeconds <= #524.seconds
			#529 panND0803counterP1 <= ND0803counterP1
			#530 panND0803counterP2 <= ND0803counterP2
			#531 workTimeN010501:TimeFromWorkTime(input: N0105workTimeP1)
			#532 panN010501workDays <= #531.days
			#533 panN010501workHours <= #531.hours
			#534 panN010501workMinutes <= #531.minutes
			#535 panN010501workSeconds <= #531.seconds
			#536 workTimeN010502:TimeFromWorkTime(input: N0105workTimeP2)
			#537 panN010502workDays <= #536.days
			#538 panN010502workHours <= #536.hours
			#539 panN010502workMinutes <= #536.minutes
			#540 panN010502workSeconds <= #536.seconds
			#541 panN0105counterP1 <= N0105counterP1
			#542 panN0105counterP2 <= N0105counterP2
			#543 workTimeN020401:TimeFromWorkTime(input: N0204workTimeP1)
			#544 panN020401workDays <= #543.days
			#545 panN020401workHours <= #543.hours
			#546 panN020401workMinutes <= #543.minutes
			#547 panN020401workSeconds <= #543.seconds
			#548 workTimeN020402:TimeFromWorkTime(input: N0204workTimeP2)
			#549 panN020402workDays <= #548.days
			#550 panN020402workHours <= #548.hours
			#551 panN020402workMinutes <= #548.minutes
			#552 panN020402workSeconds <= #548.seconds
			#553 panN0204counterP1 <= N0204counterP1
			#554 panN0204counterP2 <= N0204counterP2
			#555 workTimeN040401:TimeFromWorkTime(input: N0404workTimeP1)
			#556 panN040401workDays <= #555.days
			#557 panN040401workHours <= #555.hours
			#558 panN040401workMinutes <= #555.minutes
			#559 panN040401workSeconds <= #555.seconds
			#560 workTimeN040402:TimeFromWorkTime(input: N0404workTimeP2)
			#561 panN040402workDays <= #560.days
			#562 panN040402workHours <= #560.hours
			#563 panN040402workMinutes <= #560.minutes
			#564 panN040402workSeconds <= #560.seconds
			#565 panN0404counterP1 <= N0404counterP1
			#566 panN0404counterP2 <= N0404counterP2
			#567 workTimeUFO030101:TimeFromWorkTime(input: UFO0301workTimeP1)
			#568 panUFO030101workDays <= #567.days
			#569 panUFO030101workHours <= #567.hours
			#570 panUFO030101workMinutes <= #567.minutes
			#571 panUFO030101workSeconds <= #567.seconds
			#572 workTimeUFO030102:TimeFromWorkTime(input: UFO0301workTimeP2)
			#573 panUFO030102workDays <= #572.days
			#574 panUFO030102workHours <= #572.hours
			#575 panUFO030102workMinutes <= #572.minutes
			#576 panUFO030102workSeconds <= #572.seconds
			#577 panUFO0301counterP1 <= UFO0301counterP1
			#578 panUFO0301counterP2 <= UFO0301counterP2
		END_MACRO
		#579 panVolumeToRegen <= volumeToRegen
	END_MACRO
	#580 MACRO PSB регистры на передачу в панель (отображение)()
		(* PSB регистры на передачу в панель (отображение) *)
		#581 MACRO 8 bit output module 1()
			#582 panStartND050201 <= DD4_DO.4
			#583 panStartND050202 <= DD4_DO.5
			#584 panStartND060201 <= DD4_DO.6
			#585 panStartND060202 <= DD4_DO.7
			#586 panStartND060301 <= DD4_DO.8
			#587 panStartND060302 <= DD4_DO.9
			#588 panStartM0604 <= DD5_DI.21
			#589 panStartND070301 <= DD4_DO.10
		END_MACRO
		#590 MACRO 8 bit output module 2()
			#591 panStartND070302 <= DD4_DO.11
			#592 panStartM0702 <= DD5_DI.23
			#593 panStartND080301 <= DD1_DO3
			#594 panStartND080302 <= DD1_DO4
			#595 panStartND0804 <= DD4_DO.12
			#596 panStartM0802 <= DD5_DI.25
			#597 panStartN020401 <= DD5_DI.9
			#598 panStartN020402 <= DD5_DI.10
		END_MACRO
		#599 MACRO 8 bit output module 3()
			#600 panStartN010501 <= N0105statStartedP1
			#601 panStartN010502 <= N0105statStartedP2
			#602 panCleanFS020101 <= DD6_DI.20
			#603 panCleanFS020102 <= DD6_DI.22
			#604 panCleanFS020103 <= DD6_DI.24
			#605 panCleanFS020104 <= DD6_DI.26
			#606 panCleanFS020105 <= DD6_DI.28
			#607 panCleanFS020106 <= DD6_DI.30
		END_MACRO
		#608 MACRO 8 bit output module 4()
			#609 panCleanFS020201 <= DD7_DI. 0
			#610 panCleanFS020202 <= DD7_DI. 2
			#611 panCleanFS020203 <= DD7_DI. 4
			#612 panCleanFS020204 <= DD7_DI. 6
			#613 panCleanFS020205 <= DD7_DI. 8
			#614 panCleanFS020206 <= DD7_DI. 10
			#615 panSludgeReady <= DD7_DI.15
			#616 panStartN0401 <= DD7_DI.13
		END_MACRO
		#617 MACRO 8 bit output module 5()
			#618 panKSHE0401open <= DD9_DI.2
			#619 panFPKready <= DD7_DI.12
			#620 panFPKneedToClean <= FPKneedToClean
			#621 panStartN040401 <= DD5_DI.16
			#622 panStartN040402 <= DD5_DI.17
			#623 panStartUFO030101 <= statusUFO030101started
			#624 panStartUFO030102 <= statusUFO030102started
			#625 panAlarm <= alarm
		END_MACRO
		#626 MACRO 8 bit output module 6()
			#627 panErrorTempSensor <= DD1_AI0_error
			#628 panErrorFT0101 <= DD1_AI1_error
			#629 panErrorFT0102 <= DD1_AI2_error
			#630 panErrorQE0102 <= DD1_AI3_error
			#631 panErrorQE0102 <= DD1_AI4_error
			#632 panAlarmHighTemp <= alarmHighTemperature
			#633 panAlarmLowTemp <= alarmLowTemperature
			#634 panND0502dosingError <= ND0502dosingError
		END_MACRO
		#635 MACRO 8 bit output module 7()
			#636 panND0602dosingError <= ND0602dosingError
			#637 panND0603dosingError <= ND0603dosingError
			#638 panND0803dosingError <= ND0803dosingError
			#639 panND0804dosingError <= ND0804dosingError
			#640 panND080301emptyAlarm <= DD1_DI6
			#641 panND080302emptyAlarm <= DD1_DI7
			#642 panN010501alarm <= N010501alarm
			#643 panN010502alarm <= N010502alarm
		END_MACRO
		#644 MACRO 8 bit output module 8()
			#645 panZDE0225errorToOpen <= ZDE0225errorToOpen
			#646 panZDE0225errorToClose <= ZDE0225errorToClose
			#647 panFPKalarm <= DD7_DI.14
			#648 panFPKnotStarted <= FPKnotStarted
			#649 panErrorFPKsensor <= DD1_AI5_error
			#650 panFPKkshe0401errorToOpen <= FPKkshe0401errorToOpen
			#651 panFPKkshe0401errorToClose <= FPKkshe0401errorToClose
			#652 panUFO030101alarm <= statusUFO030101alarm
		END_MACRO
		#653 MACRO 8 bit output module 9()
			#654 panUFO030102alarm <= statusUFO030102alarm
			#655 panFilterFailToRegen020101 <= filterFailToRegen020101
			#656 panErrorToOpenZD0201 <= errorToOpenZD0201
			#657 panErrorToCloseZD0201 <= errorToCloseZD0201
			#658 panErrorToOpenZD0207 <= errorToOpenZD0207
			#659 panErrorToCloseZD0207 <= errorToCloseZD0207
			#660 panFilterFailToRegen020102 <= filterFailToRegen020102
			#661 panErrorToOpenZD0202 <= errorToOpenZD0202
		END_MACRO
		#662 MACRO 8 bit output module 10()
			#663 panErrorToCloseZD0202 <= errorToCloseZD0202
			#664 panErrorToOpenZD0208 <= errorToOpenZD0208
			#665 panErrorToCloseZD0208 <= errorToCloseZD0208
			#666 panFilterFailToRegen020103 <= filterFailToRegen020103
			#667 panErrorToOpenZD0203 <= errorToOpenZD0203
			#668 panErrorToCloseZD0203 <= errorToCloseZD0203
			#669 panErrorToOpenZD0209 <= errorToOpenZD0209
			#670 panErrorToCloseZD0209 <= errorToCloseZD0209
		END_MACRO
		#671 MACRO 8 bit output module 11()
			#672 panFilterFailToRegen020104 <= filterFailToRegen020104
			#673 panErrorToOpenZD0204 <= errorToOpenZD0204
			#674 panErrorToCloseZD0204 <= errorToCloseZD0204
			#675 panErrorToOpenZD0210 <= errorToOpenZD0210
			#676 panErrorToCloseZD0210 <= errorToCloseZD0210
			#677 panFilterFailToRegen020105 <= filterFailToRegen020105
			#678 panErrorToOpenZD0205 <= errorToOpenZD0205
			#679 panErrorToCloseZD0205 <= errorToCloseZD0205
		END_MACRO
		#680 MACRO 8 bit output module 12()
			#681 panErrorToOpenZD0211 <= errorToOpenZD0211
			#682 panErrorToCloseZD0211 <= errorToCloseZD0211
			#683 panFilterFailToRegen020106 <= filterFailToRegen020106
			#684 panErrorToOpenZD0206 <= errorToOpenZD0206
			#685 panErrorToCloseZD0206 <= errorToCloseZD0206
			#686 panErrorToOpenZD0212 <= errorToOpenZD0212
			#687 panErrorToCloseZD0212 <= errorToCloseZD0212
			#688 panFilterFailToRegen020201 <= filterFailToRegen020201
		END_MACRO
		#689 MACRO 8 bit output module 13()
			#690 panErrorToOpenZD0213 <= errorToOpenZD0213
			#691 panErrorToCloseZD0213 <= errorToCloseZD0213
			#692 panErrorToOpenZD0219 <= errorToOpenZD0219
			#693 panErrorToCloseZD0219 <= errorToCloseZD0219
			#694 panFilterFailToRegen020202 <= filterFailToRegen020202
			#695 panErrorToOpenZD0214 <= errorToOpenZD0214
			#696 panErrorToCloseZD0214 <= errorToCloseZD0214
			#697 panErrorToOpenZD0220 <= errorToOpenZD0220
		END_MACRO
		#698 MACRO 8 bit output module 14()
			#699 panErrorToCloseZD0220 <= errorToCloseZD0220
			#700 panFilterFailToRegen020203 <= filterFailToRegen020203
			#701 panErrorToOpenZD0215 <= errorToOpenZD0215
			#702 panErrorToCloseZD0215 <= errorToCloseZD0215
			#703 panErrorToOpenZD0221 <= errorToOpenZD0221
			#704 panErrorToCloseZD0221 <= errorToCloseZD0221
			#705 panFilterFailToRegen020204 <= filterFailToRegen020204
			#706 panErrorToOpenZD0216 <= errorToOpenZD0216
		END_MACRO
		#707 MACRO 8 bit output module 15()
			#708 panErrorToCloseZD0216 <= errorToCloseZD0216
			#709 panErrorToOpenZD0222 <= errorToOpenZD0222
			#710 panErrorToCloseZD0222 <= errorToCloseZD0222
			#711 panFilterFailToRegen020205 <= filterFailToRegen020205
			#712 panErrorToOpenZD0217 <= errorToOpenZD0217
			#713 panErrorToCloseZD0217 <= errorToCloseZD0217
			#714 panErrorToOpenZD0223 <= errorToOpenZD0223
			#715 panErrorToCloseZD0223 <= errorToCloseZD0223
		END_MACRO
		#716 MACRO 8 bit output module 16()
			#717 panFilterFailToRegen020206 <= filterFailToRegen020206
			#718 panErrorToOpenZD0218 <= errorToOpenZD0218
			#719 panErrorToCloseZD0218 <= errorToCloseZD0218
			#720 panErrorToOpenZD0224 <= errorToOpenZD0224
			#721 panErrorToCloseZD0224 <= errorToCloseZD0224
			#722 panAlarmPLKnetwork <= alarmPLKnetwork
			#723 panAlarmND050201 <= alarmND050201
			#724 panAlarmND050202 <= alarmND050202
		END_MACRO
		#725 MACRO 8 bit output module 17()
			#726 panAlarmND060201 <= alarmND060201
			#727 panAlarmND060202 <= alarmND060202
			#728 panAlarmND060301 <= alarmND060301
			#729 panAlarmND060302 <= alarmND060302
			#730 panAlarmND070301 <= alarmND070301
			#731 panAlarmND070302 <= alarmND070302
			#732 panAlarmND080301 <= alarmND080301
			#733 panAlarmND080302 <= alarmND080302
		END_MACRO
		#734 MACRO 8 bit output module 18()
			#735 panAlarmND0804 <= alarmND0804
			#736 panAlarmOGM0104overload <= alarmOGM0104overload
			#737 panAlarmRCHV0203overload <= alarmRCHV0203overload
			#738 panAlarmN040402 <= alarmN040402
			#739 panAlarmN040401 <= alarmN040401
			#740 panAlarmM0604 <= alarmM0604
			#741 panAlarmM0702 <= alarmM0702
			#742 panAlarmM0802 <= alarmM0802
		END_MACRO
		#743 MACRO 8 bit output module 19()
			#744 panAlarmN020401 <= alarmN020401
			#745 panAlarmN020402 <= alarmN020402
			#746 panAlarmFS020101 <= alarmFS020101
			#747 panAlarmFS020102 <= alarmFS020102
			#748 panAlarmFS020103 <= alarmFS020103
			#749 panAlarmFS020104 <= alarmFS020104
			#750 panAlarmFS020105 <= alarmFS020105
			#751 panAlarmFS020106 <= alarmFS020106
		END_MACRO
		#752 MACRO 8 bit output module 20()
			#753 panAlarmFS020201 <= alarmFS020201
			#754 panAlarmFS020202 <= alarmFS020202
			#755 panAlarmFS020203 <= alarmFS020203
			#756 panAlarmFS020204 <= alarmFS020204
			#757 panAlarmFS020205 <= alarmFS020205
			#758 panAlarmFS020206 <= alarmFS020206
			#759 panAlarmZDE0201power <= alarmZDE0201power
			#760 panAlarmZDE0202power <= alarmZDE0202power
		END_MACRO
		#761 MACRO 8 bit output module 21()
			#762 panAlarmZDE0203power <= alarmZDE0203power
			#763 panAlarmZDE0204power <= alarmZDE0204power
			#764 panAlarmZDE0205power <= alarmZDE0205power
			#765 panAlarmZDE0206power <= alarmZDE0206power
			#766 panAlarmZDE0207power <= alarmZDE0207power
			#767 panAlarmZDE0208power <= alarmZDE0208power
			#768 panAlarmZDE0209power <= alarmZDE0209power
			#769 panAlarmZDE0210power <= alarmZDE0210power
		END_MACRO
		#770 MACRO 8 bit output module 22()
			#771 panAlarmZDE0211power <= alarmZDE0211power
			#772 panAlarmZDE0212power <= alarmZDE0212power
			#773 panAlarmZDE0213power <= alarmZDE0213power
			#774 panAlarmZDE0214power <= alarmZDE0214power
			#775 panAlarmZDE0215power <= alarmZDE0215power
			#776 panAlarmZDE0216power <= alarmZDE0216power
			#777 panAlarmZDE0217power <= alarmZDE0217power
			#778 panAlarmZDE0218power <= alarmZDE0218power
		END_MACRO
		#779 MACRO 8 bit output module 23()
			#780 panAlarmZDE0219power <= alarmZDE0219power
			#781 panAlarmZDE0220power <= alarmZDE0220power
			#782 panAlarmZDE0221power <= alarmZDE0221power
			#783 panAlarmZDE0222power <= alarmZDE0222power
			#784 panAlarmZDE0223power <= alarmZDE0223power
			#785 panAlarmZDE0224power <= alarmZDE0224power
			#786 panAlarmZDE0225power <= alarmZDE0225power
			#787 panAlarmKSHE0401power <= alarmKSHE0401power
		END_MACRO
		#788 MACRO 8 bit output module 24()
			#789 panAlarmKNS <= alarmKNS
			#790 panAlarmPowerSocketFS <= alarmPowerSocketFS
			#791 panAlarmKEMvalvesPower <= alarmKEMvalvesPower
			#792 panAlarmEmergencyPressed <= alarmEmergencyPressed
			#793 panAlarmRKF <= alarmRKF
			#794 panUFO0301noFlowAttention <= UFO0301noFlowAttention
			#795 panM0604attention <= M0604attention
			#796 panM0702attention <= M0702attention
		END_MACRO
		#797 MACRO 8 bit output module 25()
			#798 panM0802attention <= M0802attention
			#799 panStatusKNS <= DD6_DI.8
			#800 panND0502statRegimeP1M <= ND0502statRegimeP1M
			#801 panND0502statRegimeP2M <= ND0502statRegimeP2M
			#802 panND0502statRegimeByC <= ND0502statRegimeByC
			#803 panND0502statRegimeByWT <= ND0502statRegimeByWT
			#804 panND0602statRegimeP1M <= ND0602statRegimeP1M
			#805 panND0602statRegimeP2M <= ND0602statRegimeP2M
		END_MACRO
		#806 MACRO 8 bit output module 26()
			#807 panND0602statRegimeByC <= ND0602statRegimeByC
			#808 panND0602statRegimeByWT <= ND0602statRegimeByWT
			#809 panND0603statRegimeP1M <= ND0603statRegimeP1M
			#810 panND0603statRegimeP2M <= ND0603statRegimeP2M
			#811 panND0603statRegimeByC <= ND0603statRegimeByC
			#812 panND0603statRegimeByWT <= ND0603statRegimeByWT
			#813 panND0703statRegimeP1M <= ND0703statRegimeP1M
			#814 panND0703statRegimeP2M <= ND0703statRegimeP2M
		END_MACRO
		#815 MACRO 8 bit output module 27()
			#816 panND0703statRegimeByC <= ND0703statRegimeByC
			#817 panND0703statRegimeByWT <= ND0703statRegimeByWT
			#818 panND0803statRegimeP1M <= ND0803statRegimeP1M
			#819 panND0803statRegimeP2M <= ND0803statRegimeP2M
			#820 panND0803statRegimeByC <= ND0803statRegimeByC
			#821 panND0803statRegimeByWT <= ND0803statRegimeByWT
			#822 panN0105statRegimeP1M <= N0105statRegimeP1M
			#823 panN0105statRegimeP2M <= N0105statRegimeP2M
		END_MACRO
		#824 MACRO 8 bit output module 28()
			#825 panN0105statRegimeByC <= N0105statRegimeByC
			#826 panN0105statRegimeByWT <= N0105statRegimeByWT
			#827 panN0204statRegimeP1M <= N0204statRegimeP1M
			#828 panN0204statRegimeP2M <= N0204statRegimeP2M
			#829 panN0204statRegimeByC <= N0204statRegimeByC
			#830 panN0204statRegimeWT <= N0204statRegimeWT
			#831 panN0404statRegimeP1M <= N0404statRegimeP1M
			#832 panN0404statRegimeP2M <= N0404statRegimeP2M
		END_MACRO
		#833 MACRO 8 bit output module 29()
			#834 panN0404statRegimeByC <= N0404statRegimeByC
			#835 panN0404statRegimeWT <= N0404statRegimeWT
			#836 panUFO0301statRegimeP1M <= UFO0301statRegimeP1M
			#837 panUFO0301statRegimeP2M <= UFO0301statRegimeP2M
			#838 panUFO0301statRegimeByC <= UFO0301statRegimeByC
			#839 panUFO0301statRegimeWT <= UFO0301statRegimeWT
			#840 panZDE0225open <= DD9_DI.0
			#841 panZDE0201open <= DD7_DI.16
		END_MACRO
		#842 MACRO 8 bit output module 30()
			#843 panZDE0201close <= DD7_DI.17
			#844 panZDE0202open <= DD7_DI.18
			#845 panZDE0202close <= DD7_DI.19
			#846 panZDE0203open <= DD7_DI.20
			#847 panZDE0203close <= DD7_DI.21
			#848 panZDE0204open <= DD7_DI.22
			#849 panZDE0204close <= DD7_DI.23
			#850 panZDE0205open <= DD7_DI.24
		END_MACRO
		#851 MACRO 8 bit output module 31()
			#852 panZDE0205close <= DD7_DI.25
			#853 panZDE0206open <= DD7_DI.26
			#854 panZDE0206close <= DD7_DI.27
			#855 panZDE0207open <= DD7_DI.28
			#856 panZDE0207close <= DD7_DI.29
			#857 panZDE0208open <= DD7_DI.30
			#858 panZDE0208close <= DD7_DI.31
			#859 panZDE0209open <= DD8_DI.0
		END_MACRO
		#860 MACRO 8 bit output module 32()
			#861 panZDE0209close <= DD8_DI.1
			#862 panZDE0210open <= DD8_DI.2
			#863 panZDE0210close <= DD8_DI.3
			#864 panZDE0211open <= DD8_DI.4
			#865 panZDE0211close <= DD8_DI.5
			#866 panZDE0212open <= DD8_DI.6
			#867 panZDE0212close <= DD8_DI.7
			#868 panZDE0213open <= DD8_DI.8
		END_MACRO
		#869 MACRO 8 bit output module 33()
			#870 panZDE0213close <= DD8_DI.9
			#871 panZDE0214open <= DD8_DI.10
			#872 panZDE0214close <= DD8_DI.11
			#873 panZDE0215open <= DD8_DI.12
			#874 panZDE0215close <= DD8_DI.13
			#875 panZDE0216open <= DD8_DI.14
			#876 panZDE0216close <= DD8_DI.15
			#877 panZDE0217open <= DD8_DI.16
		END_MACRO
		#878 MACRO 8 bit output module 34()
			#879 panZDE0217close <= DD8_DI.17
			#880 panZDE0218open <= DD8_DI.18
			#881 panZDE0218close <= DD8_DI.19
			#882 panZDE0219open <= DD8_DI.20
			#883 panZDE0219close <= DD8_DI.21
			#884 panZDE0220open <= DD8_DI.22
			#885 panZDE0220close <= DD8_DI.23
			#886 panZDE0221open <= DD8_DI.24
		END_MACRO
		#887 MACRO 8 bit output module 35()
			#888 panZDE0221close <= DD8_DI.25
			#889 panZDE0222open <= DD8_DI.26
			#890 panZDE0222close <= DD8_DI.27
			#891 panZDE0223open <= DD8_DI.28
			#892 panZDE0223close <= DD8_DI.29
			#893 panZDE0224open <= DD8_DI.30
			#894 panZDE0224close <= DD8_DI.31
			#895 panZDE0225close <= DD9_DI.1
		END_MACRO
		#896 MACRO 8 bit output module 36x()
			#897 panKSHE0401close <= DD9_DI.3
			#898 panZDE0301open <= DD1_DI12
			#899 panZDE0301close <= DD1_DI13
			#900 panZDE0302open <= DD1_DI14
			#901 panZDE0302close <= DD1_DI15
			#902 panErrorToOpenZDE0301 <= errorToOpenZDE0301
			#903 panErrorToCloseZDE0301 <= errorToCloseZDE0301
			#904 panErrorToOpenZDE0302 <= errorToOpenZDE0302
		END_MACRO
		#905 panErrorToCloseZDE0302 <= errorToCloseZDE0302
		#906 panAlarmZDE0301power <= alarmZDE0301power
		#907 panAlarmZDE0302power <= alarmZDE0302power
		#908 panUFO030101danger <= statusUFO030101danger
		#909 panUFO030102danger <= statusUFO030102danger
		#910 panUFO030101distantMode <= statusUFO030101distantMode
		#911 panUFO030102distantMode <= statusUFO030102distantMode
	END_MACRO
	#912 MACRO PFW регистры на чтение из панели (управление ПЛК)()
		#913 MUL(panTimeToOpenCloseValve, 1000)
		#914 REAL_TO_TIME(#913)
		#915 TimeToOpenCloseValve <= #914
		#916 maxTemperature <= panMaxTemperature
		#917 minTemperature <= panMinTemperature
		#918 ND0502setMaxDosVal <= panND0502setMaxDosVal
		#919 ND0502setKoefProp <= panND0502setKoefProp
		#920 ND0602setMaxDosVal <= panND0602setMaxDosVal
		#921 ND0602setKoefProp <= panND0602setKoefProp
		#922 ND0603setMaxDosVal <= panND0603setMaxDosVal
		#923 ND0603setKoefProp <= panND0603setKoefProp
		#924 ND0703pHsetValue <= panND0703pHsetValue
		#925 ND0703YoutManual <= panND0703YoutManual
		#926 ND0703koeffI <= panND0703koeffI
		#927 ND0703koeffD <= panND0703koeffD
		#928 ND0703koeffP <= panND0703koeffP
		#929 ND0803setMaxDosVal <= panND0803setMaxDosVal
		#930 ND0803setKoefProp <= panND0803setKoefProp
		#931 ND0804doseValue <= panND0804doseValue
		#932 N0105flowSetValue <= panN0105flowSetValue
		#933 N0105YoutManual <= panN0105YoutManual
		#934 N0105koeffI <= panN0105koeffI
		#935 N0105koeffD <= panN0105koeffD
		#936 N0105koeffP <= panN0105koeffP
		#937 FQS0301impulsValue <= panFQS0301impulsValue
		#938 FQS0301correction <= panFQS0301correction
		#939 MUL(panFPKtimeToWork, 1000)
		#940 REAL_TO_TIME(#939)
		#941 FPKtimeToWork <= #940
		#942 MUL(panFPKnotStartedTime, 1000)
		#943 REAL_TO_TIME(#942)
		#944 FPKnotStartedTime <= #943
		#945 FPKmaxPressureValue <= panFPKmaxPressureValue
		#946 filterValueToRegen <= panFilterValueToRegen
	END_MACRO
	#947 MACRO PSB регистры на чтение из панели (управление ПЛК)()
		(* PSB регистры на чтение из панели (управление ПЛК) *)
		#948 MACRO 8 bit input module 1()
			#949 alarmReset <= panAlarmResetButton
			#950 ND0502resetCountP1 <= panND0502resetCountP1
			#951 ND0502resetCountP2 <= panND0502resetCountP2
			#952 ND0502resetWorkTimeP1 <= panND0502resetWorkTimeP1
			#953 ND0502resetWorkTimeP2 <= panND0502resetWorkTimeP2
			#954 ND0502regimeP1M <= panND0502regimeP1M
			#955 ND0502regimeP2M <= panND0502regimeP2M
			#956 ND0502regimeByC <= panND0502regimeByC
		END_MACRO
		#957 MACRO 8 bit input module 2()
			#958 ND0502regimeByWT <= panND0502regimeByWT
			#959 ND0602resetCountP1 <= panND0602resetCountP1
			#960 ND0602resetCountP2 <= panND0602resetCountP2
			#961 ND0602resetWorkTimeP1 <= panND0602resetWorkTimeP1
			#962 ND0602resetWorkTimeP2 <= panND0602resetWorkTimeP2
			#963 ND0602regimeP1M <= panND0602regimeP1M
			#964 ND0602regimeP2M <= panND0602regimeP2M
			#965 ND0602regimeByC <= panND0602regimeByC
		END_MACRO
		#966 MACRO 8 bit input module 3()
			#967 ND0602regimeByWT <= panND0602regimeByWT
			#968 ND0603resetCountP1 <= panND0603resetCountP1
			#969 ND0603resetCountP2 <= panND0603resetCountP2
			#970 ND0603resetWorkTimeP1 <= panND0603resetWorkTimeP1
			#971 ND0603resetWorkTimeP2 <= panND0603resetWorkTimeP2
			#972 ND0603regimeP1M <= panND0603regimeP1M
			#973 ND0603regimeP2M <= panND0603regimeP2M
			#974 ND0603regimeByC <= panND0603regimeByC
		END_MACRO
		#975 MACRO 8 bit input module 4()
			#976 ND0603regimeByWT <= panND0603regimeByWT
			#977 ND0703resetCountP1 <= panND0703resetCountP1
			#978 ND0703resetCountP2 <= panND0703resetCountP2
			#979 ND0703resetWorkTimeP1 <= panND0703resetWorkTimeP1
			#980 ND0703resetWorkTimeP2 <= panND0703resetWorkTimeP2
			#981 ND0703regimeP1M <= panND0703regimeP1M
			#982 ND0703regimeP2M <= panND0703regimeP2M
			#983 ND0703regimeByC <= panND0703regimeByC
		END_MACRO
		#984 MACRO 8 bit input module 5()
			#985 ND0703regimeByWT <= panND0703regimeByWT
			#986 ND0703YmanAuto <= panND0703YmanAuto
			#987 ND0803resetCountP1 <= panND0803resetCountP1
			#988 ND0803resetCountP2 <= panND0803resetCountP2
			#989 ND0803resetWorkTimeP1 <= panND0803resetWorkTimeP1
			#990 ND0803resetWorkTimeP2 <= panND0803resetWorkTimeP2
			#991 ND0803regimeP1M <= panND0803regimeP1M
			#992 ND0803regimeP2M <= panND0803regimeP2M
		END_MACRO
		#993 MACRO 8 bit input module 6()
			#994 ND0803regimeByC <= panND0803regimeByC
			#995 ND0803regimeByWT <= panND0803regimeByWT
			#996 N0105resetCountP1 <= panN0105resetCountP1
			#997 N0105resetCountP2 <= panN0105resetCountP2
			#998 N0105resetWorkTimeP1 <= panN0105resetWorkTimeP1
			#999 N0105resetWorkTimeP2 <= panN0105resetWorkTimeP2
			#1000 N0105regimeByC <= panN0105regimeByC
			#1001 N0105regimeByWT <= panN0105regimeByWT
		END_MACRO
		#1002 MACRO 8 bit input module 7()
			#1003 N0105YmanAuto <= panN0105YmanAuto
			#1004 N0204resetCountP1 <= panN0204resetCountP1
			#1005 N0204resetCountP2 <= panN0204resetCountP2
			#1006 N0204resetWorkTimeP1 <= panN0204resetWorkTimeP1
			#1007 N0204resetWorkTimeP2 <= panN0204resetWorkTimeP2
			#1008 N0204regimeP1M <= panN0204regimeP1M
			#1009 N0204regimeP2M <= panN0204regimeP2M
			#1010 N0204regimeByC <= panN0204regimeByC
		END_MACRO
		#1011 MACRO 8 bit input module 8()
			#1012 N0204regimeWT <= panN0204regimeWT
			#1013 UFO0301resetCountP1 <= panUFO0301resetCountP1
			#1014 UFO0301resetCountP2 <= panUFO0301resetCountP2
			#1015 UFO0301resetWorkTimeP1 <= panUFO0301resetWorkTimeP1
			#1016 UFO0301resetWorkTimeP2 <= panUFO0301resetWorkTimeP2
			#1017 UFO0301regimeP1M <= panUFO0301regimeP1M
			#1018 UFO0301regimeP2M <= panUFO0301regimeP2M
			#1019 UFO0301regimeByC <= panUFO0301regimeByC
		END_MACRO
		#1020 MACRO 8 bit input module 9()
			#1021 UFO0301regimeWT <= panUFO0301regimeWT
			#1022 N0404resetCountP1 <= panN0404resetCountP1
			#1023 N0404resetCountP2 <= panN0404resetCountP2
			#1024 N0404resetWorkTimeP1 <= panN0404resetWorkTimeP1
			#1025 N0404resetWorkTimeP2 <= panN0404resetWorkTimeP2
			#1026 N0404regimeP1M <= panN0404regimeP1M
			#1027 N0404regimeP2M <= panN0404regimeP2M
			#1028 N0404regimeByC <= panN0404regimeByC
		END_MACRO
		#1029 MACRO 8 bit input module 10-11()
			(* одули 10 и 11 заполнены переменными для тестирования задвижек. / Здесь они не показаны, т.к. спешка. / Они вставлены напрямую в макросы управления промывкой фильтров. / testValvesFS020101 - testValvesFS020206 (PSB612-623) *)
			#1030 N0404regimeWT <= panN0404regimeWT
			#1031 FQS0301reset <= panFQS0301reset
			#1032 FQS0301addCorrection <= panFQS0301addCorrection
			#1033 FQS0301deleteCorrection <= panFQS0301deleteCorrection
		END_MACRO
		#1034 testKSHE0401 <= panTestKSHE0401
		#1035 testZDE0225 <= panTestZDE0225
		#1036 testZDE03 <= panTestZDE03
		#1037 manualZDE0301 <= panManualZDE0301
		#1038 manualZDE0302 <= panManualZDE0302
	END_MACRO
END_MACRO
#1039 NOT(DD6_DI.13)
#1040 alarmRCHV0203overload <= #1039
#1041 NOT(DD9_DI.5)
#1042 alarmZDE0202power <= #1041
#1043 NOT(DD9_DI.26)
#1044 alarmZDE0223power <= #1043
#1045 MACRO переменные на диспетчеризацию()
	#1046 remFT0101value <= DD1_AI1_FT0101value
	#1047 remFQS0301totalAmount <= FQS0301totalAmount
	#1048 remTemperatureValue <= temperatureValue
	#1049 remStatusN010501started <= N0105statStartedP1
	#1050 remStatusN010502started <= N0105statStartedP2
	#1051 remStatusUFO030101started <= statusUFO030101started
	#1052 remStatusUFO030102started <= statusUFO030102started
	#1053 remAlarm <= Alarm
	#1054 remN010501alarm <= N010501alarm
	#1055 remN010502alarm <= N010502alarm
	#1056 remFPKalarm <= DD7_DI.14
	#1057 remUFO030101alarm <= statusUFO030101alarm
	#1058 remUFO030102alarm <= statusUFO030102alarm
	#1059 remAlarmEmergencyPressed <= alarmEmergencyPressed
	#1060 remAlarmOOGM0104overload <= DD6_DI.11
	#1061 remAlarmRCHV0203overload <= DD6_DI.13
END_MACRO
#1062 NOT(DD5_DI.14)
#1063 alarmN040402 <= #1062
#1064 NOT(DD9_DI.6)
#1065 alarmZDE0203power <= #1064
#1066 NOT(DD9_DI.27)
#1067 alarmZDE0224power <= #1066
#1068 NOT(DD5_DI.15)
#1069 alarmN040401 <= #1068
#1070 NOT(DD9_DI.7)
#1071 alarmZDE0204power <= #1070
#1072 NOT(DD9_DI.28)
#1073 alarmZDE0225power <= #1072
#1074 NOT(DD5_DI.20)
#1075 alarmM0604 <= #1074
#1076 NOT(DD9_DI.8)
#1077 alarmZDE0205power <= #1076
#1078 NOT(DD9_DI.29)
#1079 alarmKSHE0401power <= #1078
#1080 NOT(DD5_DI.22)
#1081 alarmM0702 <= #1080
#1082 NOT(DD9_DI.9)
#1083 alarmZDE0206power <= #1082
#1084 NOT(DD6_DI.9)
#1085 alarmKNS <= #1084
#1086 NOT(DD5_DI.24)
#1087 alarmM0802 <= #1086
#1088 NOT(DD9_DI.10)
#1089 alarmZDE0207power <= #1088
#1090 NOT(DD6_DI.17)
#1091 alarmPowerSocketFS <= #1090
#1092 NOT(DD5_DI.7)
#1093 alarmN020401 <= #1092
#1094 NOT(DD9_DI.11)
#1095 alarmZDE0208power <= #1094
#1096 NOT(DD6_DI.18)
#1097 alarmKEMvalvesPower <= #1096
#1098 NOT(DD5_DI.8)
#1099 alarmN020402 <= #1098
#1100 NOT(DD9_DI.12)
#1101 alarmZDE0209power <= #1100
#1102 NOT(DD1_DI4)
#1103 alarmEmergencyPressed <= #1102
#1104 GT(DD1_AI2_FT0102value, 0)
#1105 filterPulserGen:PulsePerSec(start: #1104)
#1106 DIV(DD1_AI2_FT0102value, 3600)
#1107 ADD(EN: #1105.out, #1106, filterTotalAmountFT0102)
#1108 filterTotalAmountFT0102 <= #1107
#1109 NOT(DD6_DI.21)
#1110 alarmFS020101 <= #1109
#1111 NOT(DD9_DI.13)
#1112 alarmZDE0210power <= #1111
#1113 NOT(DD1_DI5)
#1114 alarmRKF <= #1113
#1115 NOT(DD9_DI.30)
#1116 alarmZDE0301power <= #1115
#1117 NOT(DD9_DI.31)
#1118 alarmZDE0302power <= #1117
#1119 MOVE(EN: filterTotalAmountReset, 0)
#1120 filterTotalAmountFT0102 <= #1119
#1121 SUB(filterValueToRegen, filterTotalAmountFT0102)
#1122 volumeToRegen <= #1121
#1123 GE(filterTotalAmountFT0102, filterValueToRegen)
#1124 MACRO управление промывкой фильтра ФС02.01.01(pin 1 "сигнал на промывку": #1123, pin 2 "авария фильтра": DD6_DI.21, pin 3 "подтверждение промывки": DD6_DI.20, pin 4 "сброс аварий": alarmReset, pin 5 "начать очередь снова": filterStartNewQueue, pin 6 "ЗДЭ02.01 открыта": DD7_DI.16, pin 7 "ЗДЭ02.01 закрыта": DD7_DI.17, pin 8 "ЗДЭ02.07 открыта": DD7_DI.28, pin 9 "ЗДЭ02.07 закрыта": DD7_DI.29, pin 10 "время движения ЗДЭ": timeToOpenCloseValve, pin 11 "авария питания ЗДЭ02.01": DD9_DI.4, pin 12 "авария питания ЗДЭ02.07": DD9_DI.10)
	(* если открыт = фильтрация *)
	(* если открыт = промывка *)
	(* <- выход использовать в / последнем фильтре для / начала очереди заново *)
	out 1 "следующий в очереди" <= #1127.output
	out 2 "промыть ФС02.01.01" <= #1126
	#1125 ZD0201:SimpleValve(inputOpen: NOT #1126, inputClose: #1126, statusOpen: pin 6, statusClose: pin 7, reset: pin 4, timeToOpenClose: pin 10)
	out 6 "открыть ЗДЭ02.01" <= #1125.outputOpen
	out 7 "закрыть ЗДЭ02.01" <= #1125.outputClose
	out 8 "авария открытия ЗДЭ02.01" <= #1125.errorToOpen
	#1126 OR(panTestValvesFS020101, #1127.regenFilterOUT)
	out 9 "авария закрытия ЗДЭ02.01" <= #1125.errorToClose
	#1127 FS020101manager:FilterQueueManager(input: pin 1, filterAlarm: #1128, regenFilterStatus: pin 3, alarmReset: pin 4, startNextLoop: pin 5)
	#1128 OR(alarmZD020107, pin 2, pin 11, pin 12)
	out 3 "ФС02.01.01 промыт" <= #1127.regenerated
	out 4 "не удалось промыть" <= #1127.failToRegen
	#1129 OR(#1125.errorToOpen, #1125.errorToClose, #1131.errorToOpen, #1131.errorToClose)
	#1130 alarmZD020107 <= #1129
	out 5 "сброс счетчика" <= #1127.counterReset
	#1131 ZD0207:SimpleValve(inputOpen: #1126, inputClose: NOT #1126, statusOpen: pin 8, statusClose: pin 9, reset: pin 4, timeToOpenClose: pin 10)
	out 10 "открыть ЗДЭ02.07" <= #1131.outputOpen
	out 11 "закрыть ЗДЭ02.07" <= #1131.outputClose
	out 12 "авария открытия ЗДЭ02.07" <= #1131.errorToOpen
	out 13 "авария закрытия ЗДЭ02.07" <= #1131.errorToClose
END_MACRO
#1132 DD2_DO.4 <= #1124.out 2
#1133 regeneratedFS020101 <= #1124.out 3
#1134 filterFailToRegen020101 <= #1124.out 4
#1135 filterTotalAmountReset <= #1124.out 5
#1136 DD2_DO.16 <= #1124.out 6
#1137 DD2_DO.17 <= #1124.out 7
#1138 errorToOpenZD0201 <= #1124.out 8
#1139 errorToCloseZD0201 <= #1124.out 9
#1140 DD2_DO.28 <= #1124.out 10
#1141 DD2_DO.29 <= #1124.out 11
#1142 errorToOpenZD0207 <= #1124.out 12
#1143 errorToCloseZD0207 <= #1124.out 13
#1144 MACRO управление промывкой фильтра ФС02.01.02(pin 1 "сигнал на промывку": #1124.out 1, pin 2 "авария фильтра": DD6_DI.23, pin 3 "подтверждение промывки": DD6_DI.22, pin 4 "сброс аварий": alarmReset, pin 5 "начать очередь снова": filterStartNewQueue, pin 6 "ЗДЭ02.02 открыта": DD7_DI.18, pin 7 "ЗДЭ02.02 закрыта": DD7_DI.19, pin 8 "ЗДЭ02.08 открыта": DD7_DI.30, pin 9 "ЗДЭ02.08 закрыта": DD7_DI.31, pin 10 "время движения ЗДЭ": timeToOpenCloseValve, pin 11 "авария питания ЗДЭ02.02": DD9_DI.5, pin 12 "авария питания ЗДЭ02.08": DD9_DI.11)
	(* если открыт = фильтрация *)
	(* если открыт = промывка *)
	(* <- выход использовать в / последнем фильтре для / начала очереди заново *)
	out 1 "следующий в очереди" <= #1147.output
	out 2 "промыть ФС02.01.02" <= #1146
	#1145 ZD0202:SimpleValve(inputOpen: NOT #1146, inputClose: #1146, statusOpen: pin 6, statusClose: pin 7, reset: pin 4, timeToOpenClose: pin 10)
	out 5 "открыть ЗДЭ02.02" <= #1145.outputOpen
	out 6 "закрыть ЗДЭ02.02" <= #1145.outputClose
	out 7 "авария открытия ЗДЭ02.02" <= #1145.errorToOpen
	#1146 OR(panTestValvesFS020102, #1147.regenFilterOUT)
	out 8 "авария закрытия ЗДЭ02.02" <= #1145.errorToClose
	#1147 FS020102manager:FilterQueueManager(input: pin 1, filterAlarm: #1148, regenFilterStatus: pin 3, alarmReset: pin 4, startNextLoop: pin 5)
	#1148 OR(alarmZD020208, pin 2, pin 11, pin 12)
	#1149 OR(#1145.errorToOpen, #1145.errorToClose, #1151.errorToOpen, #1151.errorToClose)
	#1150 alarmZD020208 <= #1149
	out 3 "ФС02.01.02 промыт" <= #1147.regenerated
	out 4 "не удалось промыть" <= #1147.failToRegen
	#1151 ZD0208:SimpleValve(inputOpen: #1146, inputClose: NOT #1146, statusOpen: pin 8, statusClose: pin 9, reset: pin 4, timeToOpenClose: pin 10)
	out 9 "открыть ЗДЭ02.08" <= #1151.outputOpen
	out 10 "закрыть ЗДЭ02.08" <= #1151.outputClose
	out 11 "авария открытия ЗДЭ02.08" <= #1151.errorToOpen
	out 12 "авария закрытия ЗДЭ02.08" <= #1151.errorToClose
END_MACRO
#1152 DD2_DO.5 <= #1144.out 2
#1153 regeneratedFS020102 <= #1144.out 3
#1154 filterFailToRegen020102 <= #1144.out 4
#1155 DD2_DO.18 <= #1144.out 5
#1156 DD2_DO.19 <= #1144.out 6
#1157 errorToOpenZD0202 <= #1144.out 7
#1158 errorToCloseZD0202 <= #1144.out 8
#1159 DD2_DO.30 <= #1144.out 9
#1160 DD2_DO.31 <= #1144.out 10
#1161 errorToOpenZD0208 <= #1144.out 11
#1162 errorToCloseZD0208 <= #1144.out 12
#1163 MACRO управление промывкой фильтра ФС02.01.03(pin 1 "сигнал на промывку": #1144.out 1, pin 2 "авария фильтра": DD6_DI.25, pin 3 "подтверждение промывки": DD6_DI.24, pin 4 "сброс аварий": alarmReset, pin 5 "начать очередь снова": filterStartNewQueue, pin 6 "ЗДЭ02.03 открыта": DD7_DI.20, pin 7 "ЗДЭ02.03 закрыта": DD7_DI.21, pin 8 "ЗДЭ02.09 открыта": DD8_DI.0, pin 9 "ЗДЭ02.09 закрыта": DD8_DI.1, pin 10 "время движения ЗДЭ": timeToOpenCloseValve, pin 11 "авария питания ЗДЭ02.03": DD9_DI.6, pin 12 "авария питания ЗДЭ02.09": DD9_DI.12)
	(* если открыт = фильтрация *)
	(* если открыт = промывка *)
	(* <- выход использовать в / последнем фильтре для / начала очереди заново *)
	out 1 "следующий в очереди" <= #1166.output
	out 2 "промыть ФС02.01.03" <= #1165
	#1164 ZD0203:SimpleValve(inputOpen: NOT #1165, inputClose: #1165, statusOpen: pin 6, statusClose: pin 7, reset: pin 4, timeToOpenClose: pin 10)
	out 5 "открыть ЗДЭ02.03" <= #1164.outputOpen
	out 6 "закрыть ЗДЭ02.03" <= #1164.outputClose
	out 7 "авария открытия ЗДЭ02.03" <= #1164.errorToOpen
	#1165 OR(panTestValvesFS020103, #1166.regenFilterOUT)
	out 8 "авария закрытия ЗДЭ02.03" <= #1164.errorToClose
	#1166 FS020103manager:FilterQueueManager(input: pin 1, filterAlarm: #1167, regenFilterStatus: pin 3, alarmReset: pin 4, startNextLoop: pin 5)
	#1167 OR(alarmZD020309, pin 2, pin 11, pin 12)
	#1168 OR(#1164.errorToOpen, #1164.errorToClose, #1170.errorToOpen, #1170.errorToClose)
	#1169 alarmZD020309 <= #1168
	out 3 "ФС02.01.03 промыт" <= #1166.regenerated
	out 4 "не удалось промыть" <= #1166.failToRegen
	#1170 ZD0209:SimpleValve(inputOpen: #1165, inputClose: NOT #1165, statusOpen: pin 8, statusClose: pin 9, reset: pin 4, timeToOpenClose: pin 10)
	out 9 "открыть ЗДЭ02.09" <= #1170.outputOpen
	out 10 "закрыть ЗДЭ02.09" <= #1170.outputClose
	out 11 "авария открытия ЗДЭ02.09" <= #1170.errorToOpen
	out 12 "авария закрытия ЗДЭ02.09" <= #1170.errorToClose
END_MACRO
#1171 DD2_DO.6 <= #1163.out 2
#1172 regeneratedFS020103 <= #1163.out 3
#1173 filterFailToRegen020103 <= #1163.out 4
#1174 DD2_DO.20 <= #1163.out 5
#1175 DD2_DO.21 <= #1163.out 6
#1176 errorToOpenZD0203 <= #1163.out 7
#1177 errorToCloseZD0203 <= #1163.out 8
#1178 DD3_DO.0 <= #1163.out 9
#1179 DD3_DO.1 <= #1163.out 10
#1180 errorToOpenZD0209 <= #1163.out 11
#1181 errorToCloseZD0209 <= #1163.out 12
#1182 MACRO управление промывкой фильтра ФС02.01.04(pin 1 "сигнал на промывку": #1163.out 1, pin 2 "авария фильтра": DD6_DI.27, pin 3 "подтверждение промывки": DD6_DI.26, pin 4 "сброс аварий": alarmReset, pin 5 "начать очередь снова": filterStartNewQueue, pin 6 "ЗДЭ02.04 открыта": DD7_DI.22, pin 7 "ЗДЭ02.04 закрыта": DD7_DI.23, pin 8 "ЗДЭ02.10 открыта": DD8_DI.2, pin 9 "ЗДЭ02.10 закрыта": DD8_DI.3, pin 10 "время движения ЗДЭ": timeToOpenCloseValve, pin 11 "авария питания ЗДЭ02.04": DD9_DI.7, pin 12 "авария питания ЗДЭ02.10": DD9_DI.13)
	(* если открыт = фильтрация *)
	(* если открыт = промывка *)
	(* <- выход использовать в / последнем фильтре для / начала очереди заново *)
	out 1 "следующий в очереди" <= #1185.output
	out 2 "промыть ФС02.01.04" <= #1184
	#1183 ZD0204:SimpleValve(inputOpen: NOT #1184, inputClose: #1184, statusOpen: pin 6, statusClose: pin 7, reset: pin 4, timeToOpenClose: pin 10)
	out 5 "открыть ЗДЭ02.04" <= #1183.outputOpen
	out 6 "закрыть ЗДЭ02.04" <= #1183.outputClose
	out 7 "авария открытия ЗДЭ02.04" <= #1183.errorToOpen
	#1184 OR(panTestValvesFS020104, #1185.regenFilterOUT)
	out 8 "авария закрытия ЗДЭ02.04" <= #1183.errorToClose
	#1185 FS020104manager:FilterQueueManager(input: pin 1, filterAlarm: #1186, regenFilterStatus: pin 3, alarmReset: pin 4, startNextLoop: pin 5)
	#1186 OR(alarmZD020410, pin 2, pin 11, pin 12)
	#1187 OR(#1183.errorToOpen, #1183.errorToClose, #1189.errorToOpen, #1189.errorToClose)
	#1188 alarmZD020410 <= #1187
	out 3 "ФС02.01.04 промыт" <= #1185.regenerated
	out 4 "не удалось промыть" <= #1185.failToRegen
	#1189 ZD0210:SimpleValve(inputOpen: #1184, inputClose: NOT #1184, statusOpen: pin 8, statusClose: pin 9, reset: pin 4, timeToOpenClose: pin 10)
	out 9 "открыть ЗДЭ02.10" <= #1189.outputOpen
	out 10 "закрыть ЗДЭ02.10" <= #1189.outputClose
	out 11 "авария открытия ЗДЭ02.10" <= #1189.errorToOpen
	out 12 "авария закрытия ЗДЭ02.10" <= #1189.errorToClose
END_MACRO
#1190 DD2_DO.7 <= #1182.out 2
#1191 regeneratedFS020104 <= #1182.out 3
#1192 filterFailToRegen020104 <= #1182.out 4
#1193 DD2_DO.22 <= #1182.out 5
#1194 DD2_DO.23 <= #1182.out 6
#1195 errorToOpenZD0204 <= #1182.out 7
#1196 errorToCloseZD0204 <= #1182.out 8
#1197 DD3_DO.2 <= #1182.out 9
#1198 DD3_DO.3 <= #1182.out 10
#1199 errorToOpenZD0210 <= #1182.out 11
#1200 errorToCloseZD0210 <= #1182.out 12
#1201 MACRO управление промывкой фильтра ФС02.01.05(pin 1 "сигнал на промывку": #1182.out 1, pin 2 "авария фильтра": DD6_DI.29, pin 3 "подтверждение промывки": DD6_DI.28, pin 4 "сброс аварий": alarmReset, pin 5 "начать очередь снова": filterStartNewQueue, pin 6 "ЗДЭ02.05 открыта": DD7_DI.24, pin 7 "ЗДЭ02.05 закрыта": DD7_DI.25, pin 8 "ЗДЭ02.11 открыта": DD8_DI.4, pin 9 "ЗДЭ02.11 закрыта": DD8_DI.5, pin 10 "время движения ЗДЭ": timeToOpenCloseValve, pin 11 "авария питания ЗДЭ02.05": DD9_DI.8, pin 12 "авария питания ЗДЭ02.11": DD9_DI.14)
	(* если открыт = фильтрация *)
	(* если открыт = промывка *)
	(* <- выход использовать в / последнем фильтре для / начала очереди заново *)
	out 1 "следующий в очереди" <= #1204.output
	out 2 "промыть ФС02.01.05" <= #1203
	#1202 ZD0205:SimpleValve(inputOpen: NOT #1203, inputClose: #1203, statusOpen: pin 6, statusClose: pin 7, reset: pin 4, timeToOpenClose: pin 10)
	out 5 "открыть ЗДЭ02.05" <= #1202.outputOpen
	out 6 "закрыть ЗДЭ02.05" <= #1202.outputClose
	out 7 "авария открытия ЗДЭ02.05" <= #1202.errorToOpen
	#1203 OR(panTestValvesFS020105, #1204.regenFilterOUT)
	out 8 "авария закрытия ЗДЭ02.05" <= #1202.errorToClose
	#1204 FS020105manager:FilterQueueManager(input: pin 1, filterAlarm: #1205, regenFilterStatus: pin 3, alarmReset: pin 4, startNextLoop: pin 5)
	#1205 OR(alarmZD020511, pin 2, pin 11, pin 12)
	#1206 OR(#1202.errorToOpen, #1202.errorToClose, #1208.errorToOpen, #1208.errorToClose)
	#1207 alarmZD020511 <= #1206
	out 3 "ФС02.01.05 промыт" <= #1204.regenerated
	out 4 "не удалось промыть" <= #1204.failToRegen
	#1208 ZD0211:SimpleValve(inputOpen: #1203, inputClose: NOT #1203, statusOpen: pin 8, statusClose: pin 9, reset: pin 4, timeToOpenClose: pin 10)
	out 9 "открыть ЗДЭ02.11" <= #1208.outputOpen
	out 10 "закрыть ЗДЭ02.11" <= #1208.outputClose
	out 11 "авария открытия ЗДЭ02.11" <= #1208.errorToOpen
	out 12 "авария закрытия ЗДЭ02.11" <= #1208.errorToClose
END_MACRO
#1209 DD2_DO.8 <= #1201.out 2
#1210 regeneratedFS020105 <= #1201.out 3
#1211 filterFailToRegen020105 <= #1201.out 4
#1212 DD2_DO.24 <= #1201.out 5
#1213 DD2_DO.25 <= #1201.out 6
#1214 errorToOpenZD0205 <= #1201.out 7
#1215 errorToCloseZD0205 <= #1201.out 8
#1216 DD3_DO.4 <= #1201.out 9
#1217 DD3_DO.5 <= #1201.out 10
#1218 errorToOpenZD0211 <= #1201.out 11
#1219 errorToCloseZD0211 <= #1201.out 12
#1220 MACRO управление промывкой фильтра ФС02.01.06(pin 1 "сигнал на промывку": #1201.out 1, pin 2 "авария фильтра": DD6_DI.31, pin 3 "подтверждение промывки": DD6_DI.30, pin 4 "сброс аварий": alarmReset, pin 5 "начать очередь снова": filterStartNewQueue, pin 6 "ЗДЭ02.06 открыта": DD7_DI.26, pin 7 "ЗДЭ02.06 закрыта": DD7_DI.27, pin 8 "ЗДЭ02.12 открыта": DD8_DI.6, pin 9 "ЗДЭ02.12 закрыта": DD8_DI.7, pin 10 "время движения ЗДЭ": timeToOpenCloseValve, pin 11 "авария питания ЗДЭ02.06": DD9_DI.9, pin 12 "авария питания ЗДЭ02.12": DD9_DI.15)
	(* если открыт = фильтрация *)
	(* если открыт = промывка *)
	(* <- выход использовать в / последнем фильтре для / начала очереди заново *)
	out 1 "следующий в очереди" <= #1223.output
	out 2 "промыть ФС02.01.06" <= #1222
	#1221 ZD0206:SimpleValve(inputOpen: NOT #1222, inputClose: #1222, statusOpen: pin 6, statusClose: pin 7, reset: pin 4, timeToOpenClose: pin 10)
	out 5 "открыть ЗДЭ02.06" <= #1221.outputOpen
	out 6 "закрыть ЗДЭ02.06" <= #1221.outputClose
	out 7 "авария открытия ЗДЭ02.06" <= #1221.errorToOpen
	#1222 OR(panTestValvesFS020106, #1223.regenFilterOUT)
	out 8 "авария закрытия ЗДЭ02.06" <= #1221.errorToClose
	#1223 FS020106manager:FilterQueueManager(input: pin 1, filterAlarm: #1224, regenFilterStatus: pin 3, alarmReset: pin 4, startNextLoop: pin 5)
	#1224 OR(alarmZD020612, pin 2, pin 11, pin 12)
	#1225 OR(#1221.errorToOpen, #1221.errorToClose, #1227.errorToOpen, #1227.errorToClose)
	#1226 alarmZD020612 <= #1225
	out 3 "ФС02.01.06 промыт" <= #1223.regenerated
	out 4 "не удалось промыть" <= #1223.failToRegen
	#1227 ZD0212:SimpleValve(inputOpen: #1222, inputClose: NOT #1222, statusOpen: pin 8, statusClose: pin 9, reset: pin 4, timeToOpenClose: pin 10)
	out 9 "открыть ЗДЭ02.12" <= #1227.outputOpen
	out 10 "закрыть ЗДЭ02.12" <= #1227.outputClose
	out 11 "авария открытия ЗДЭ02.12" <= #1227.errorToOpen
	out 12 "авария закрытия ЗДЭ02.12" <= #1227.errorToClose
END_MACRO
#1228 DD2_DO.9 <= #1220.out 2
#1229 regeneratedFS020106 <= #1220.out 3
#1230 filterFailToRegen020106 <= #1220.out 4
#1231 DD2_DO.26 <= #1220.out 5
#1232 DD2_DO.27 <= #1220.out 6
#1233 errorToOpenZD0206 <= #1220.out 7
#1234 errorToCloseZD0206 <= #1220.out 8
#1235 DD3_DO.6 <= #1220.out 9
#1236 DD3_DO.7 <= #1220.out 10
#1237 errorToOpenZD0212 <= #1220.out 11
#1238 errorToCloseZD0212 <= #1220.out 12
